LIN {X 0,Y 355.379,Z 611.91,A -85,B 0,C 180,E1 12290.278,E2 12290.278} C_VEL
LIN {X 0,Y 355.45,Z 611.91,A -85,B 0,C 180,E1 12296.376,E2 12296.376} C_VEL
LIN {X 0,Y 355.743,Z 612.609,A -85,B 0,C 180,E1 12302.347,E2 12302.347} C_VEL
LIN {X 0,Y 357.646,Z 617.074,A -85,B 0,C 180,E1 12304.424,E2 12304.424} C_VEL
LIN {X 0,Y 362.835,Z 620.735,A -85,B 0,C 180,E1 12309.929,E2 12309.929} C_VEL
LIN {X 0,Y 365.157,Z 625.028,A -85,B 0,C 180,E1 12313.368,E2 12313.368} C_VEL
LIN {X 0,Y 368.691,Z 627.214,A -85,B 0,C 180,E1 12319.387,E2 12319.387} C_VEL
LIN {X 0,Y 370.662,Z 628.317,A -85,B 0,C 180,E1 12325.314,E2 12325.314} C_VEL
LIN {X 0,Y 371.12,Z 629.145,A -85,B 0,C 180,E1 12330,E2 12330} C_VEL
LIN {X 0,Y 370.62,Z 627.699,A -85,B 0,C 180,E1 12335.127,E2 12335.127} C_VEL
LIN {X 0,Y 368.358,Z 627.102,A -85,B 0,C 180,E1 12341.241,E2 12341.241} C_VEL
LIN {X 0,Y 364.863,Z 624.711,A -85,B 0,C 180,E1 12347.042,E2 12347.042} C_VEL
LIN {X 0,Y 362.708,Z 620.111,A -85,B 0,C 180,E1 12350.279,E2 12350.279} C_VEL
LIN {X 0,Y 357.276,Z 616.633,A -85,B 0,C 180,E1 12355.924,E2 12355.924} C_VEL
LIN {X 0,Y 355.733,Z 612.233,A -85,B 0,C 180,E1 12357.698,E2 12357.698} C_VEL
LIN {X 0,Y 355.573,Z 611.91,A -85,B 0,C 180,E1 12363.611,E2 12363.611} C_VEL
LIN {X 0,Y 355.371,Z 611.91,A -85,B 0,C 180,E1 12369.921,E2 12369.921} C_VEL
LIN {X 0,Y 355.212,Z 611.91,A -85,B 0,C 180,E1 12376.997,E2 12376.997} C_VEL
LIN {X 0,Y 355.407,Z 611.91,A -85,B 0,C 180,E1 12384.038,E2 12384.038} C_VEL
LIN {X 0,Y 355.733,Z 611.91,A -85,B 0,C 180,E1 12392.08,E2 12392.08} C_VEL
LIN {X 0,Y 356.072,Z 611.91,A -85,B 0,C 180,E1 12400.109,E2 12400.109} C_VEL
LIN {X 0,Y 356.301,Z 611.91,A -85,B 0,C 180,E1 12407.784,E2 12407.784} C_VEL
LIN {X 0,Y 356.826,Z 611.91,A -85,B 0,C 180,E1 12415.128,E2 12415.128} C_VEL
LIN {X 0,Y 357.149,Z 611.91,A -85,B 0,C 180,E1 12419.996,E2 12419.996} C_VEL
LIN {X 0,Y 356.648,Z 611.91,A -85,B 0,C 180,E1 12427.312,E2 12427.312} C_VEL
LIN {X 0,Y 356.243,Z 611.91,A -85,B 0,C 180,E1 12434.769,E2 12434.769} C_VEL
LIN {X 0,Y 355.891,Z 611.91,A -85,B 0,C 180,E1 12442.507,E2 12442.507} C_VEL
LIN {X 0,Y 355.712,Z 611.91,A -85,B 0,C 180,E1 12447.912,E2 12447.912} C_VEL
LIN {X 0,Y 355.436,Z 611.91,A -85,B 0,C 180,E1 12455.968,E2 12455.968} C_VEL
LIN {X 0,Y 355.447,Z 612.191,A -85,B 0,C 180,E1 12463.097,E2 12463.097} C_VEL
LIN {X 0,Y 358.002,Z 617.714,A -85,B 0,C 180,E1 12463.686,E2 12463.686} C_VEL
LIN {X 0,Y 377.621,Z 652.126,A -85,B 0,C 180,E1 12467.658,E2 12467.658} C_VEL
LIN {X 0,Y 390.531,Z 683.879,A -85,B 0,C 180,E1 12470.83,E2 12470.83} C_VEL
LIN {X 0,Y 390.809,Z 689.821,A -85,B 0,C 180,E1 12471.237,E2 12471.237} C_VEL
LIN {X 0,Y 385.398,Z 724.931,A -85,B 0,C 180,E1 12473.37,E2 12473.37} C_VEL
LIN {X 0,Y 378.325,Z 760.211,A -85,B 0,C 180,E1 12476.611,E2 12476.611} C_VEL
LIN {X 0,Y 371.725,Z 789.157,A -85,B 0,C 180,E1 12480.406,E2 12480.406} C_VEL
LIN {X 0,Y 365.554,Z 815.678,A -85,B 0,C 180,E1 12485.206,E2 12485.206} C_VEL
LIN {X 0,Y 361.007,Z 837.123,A -85,B 0,C 180,E1 12490.726,E2 12490.726} C_VEL
LIN {X 0,Y 358.596,Z 851.842,A -85,B 0,C 180,E1 12496.164,E2 12496.164} C_VEL
LIN {X 0,Y 357.652,Z 861.108,A -85,B 0,C 180,E1 12501.479,E2 12501.479} C_VEL
LIN {X 0,Y 357.41,Z 864.984,A -85,B 0,C 180,E1 12505.14,E2 12505.14} C_VEL
LIN {X 0,Y 357.395,Z 866.804,A -85,B 0,C 180,E1 12510,E2 12510} C_VEL
LIN {X 0,Y 357.423,Z 864.984,A -85,B 0,C 180,E1 12514.86,E2 12514.86} C_VEL
LIN {X 0,Y 357.893,Z 857.822,A -85,B 0,C 180,E1 12520.716,E2 12520.716} C_VEL
LIN {X 0,Y 359.264,Z 846.967,A -85,B 0,C 180,E1 12525.875,E2 12525.875} C_VEL
LIN {X 0,Y 358.591,Z 843.692,A -85,B 0,C 180,E1 12527.166,E2 12527.166} C_VEL
LIN {X 0,Y 354.052,Z 833.781,A -85,B 0,C 180,E1 12530.653,E2 12530.653} C_VEL
LIN {X 0,Y 354.208,Z 832.758,A -85,B 0,C 180,E1 12530.967,E2 12530.967} C_VEL
LIN {X 0,Y 359.253,Z 810.976,A -85,B 0,C 180,E1 12536.265,E2 12536.265} C_VEL
LIN {X 0,Y 365.983,Z 784.072,A -85,B 0,C 180,E1 12540.966,E2 12540.966} C_VEL
LIN {X 0,Y 373.426,Z 752.301,A -85,B 0,C 180,E1 12544.887,E2 12544.887} C_VEL
LIN {X 0,Y 379.7,Z 721.122,A -85,B 0,C 180,E1 12547.605,E2 12547.605} C_VEL
LIN {X 0,Y 384.344,Z 687.397,A -85,B 0,C 180,E1 12549.682,E2 12549.682} C_VEL
LIN {X 0,Y 372.11,Z 656.453,A -85,B 0,C 180,E1 12552.922,E2 12552.922} C_VEL
LIN {X 0,Y 353.965,Z 623.815,A -85,B 0,C 180,E1 12556.821,E2 12556.821} C_VEL
LIN {X 0,Y 347.602,Z 613.745,A -85,B 0,C 180,E1 12558.246,E2 12558.246} C_VEL
LIN {X 0,Y 347.379,Z 611.91,A -85,B 0,C 180,E1 12558.537,E2 12558.537} C_VEL
LIN {X 0,Y 347.581,Z 611.91,A -85,B 0,C 180,E1 12565.857,E2 12565.857} C_VEL
LIN {X 0,Y 347.709,Z 611.91,A -85,B 0,C 180,E1 12571.388,E2 12571.388} C_VEL
LIN {X 0,Y 348.051,Z 611.91,A -85,B 0,C 180,E1 12579.64,E2 12579.64} C_VEL
LIN {X 0,Y 348.287,Z 611.91,A -85,B 0,C 180,E1 12584.886,E2 12584.886} C_VEL
LIN {X 0,Y 348.726,Z 611.91,A -85,B 0,C 180,E1 12592.521,E2 12592.521} C_VEL
LIN {X 0,Y 349.186,Z 611.91,A -85,B 0,C 180,E1 12600.005,E2 12600.005} C_VEL
LIN {X 0,Y 348.793,Z 611.91,A -85,B 0,C 180,E1 12607.487,E2 12607.487} C_VEL
LIN {X 0,Y 348.3,Z 611.91,A -85,B 0,C 180,E1 12615.123,E2 12615.123} C_VEL
LIN {X 0,Y 348.081,Z 611.91,A -85,B 0,C 180,E1 12620.368,E2 12620.368} C_VEL
LIN {X 0,Y 347.814,Z 611.91,A -85,B 0,C 180,E1 12625.809,E2 12625.809} C_VEL
LIN {X 0,Y 347.611,Z 611.91,A -85,B 0,C 180,E1 12631.516,E2 12631.516} C_VEL
LIN {X 0,Y 347.4,Z 611.91,A -85,B 0,C 180,E1 12638.327,E2 12638.327} C_VEL
LIN {X 0,Y 347.356,Z 611.91,A -85,B 0,C 180,E1 12645.781,E2 12645.781} C_VEL
LIN {X 0,Y 347.391,Z 611.91,A -85,B 0,C 180,E1 12652.398,E2 12652.398} C_VEL
LIN {X 0,Y 347.567,Z 612.488,A -85,B 0,C 180,E1 12656.155,E2 12656.155} C_VEL
LIN {X 0,Y 349.455,Z 617.075,A -85,B 0,C 180,E1 12657.916,E2 12657.916} C_VEL
LIN {X 0,Y 354.366,Z 620.607,A -85,B 0,C 180,E1 12662.05,E2 12662.05} C_VEL
LIN {X 0,Y 357.147,Z 625.381,A -85,B 0,C 180,E1 12664.917,E2 12664.917} C_VEL
LIN {X 0,Y 361.714,Z 628.59,A -85,B 0,C 180,E1 12669.782,E2 12669.782} C_VEL
LIN {X 0,Y 364.262,Z 632.973,A -85,B 0,C 180,E1 12673.475,E2 12673.475} C_VEL
LIN {X 0,Y 367.686,Z 635.044,A -85,B 0,C 180,E1 12679.321,E2 12679.321} C_VEL
LIN {X 0,Y 369.663,Z 636.06,A -85,B 0,C 180,E1 12685.154,E2 12685.154} C_VEL
LIN {X 0,Y 370.158,Z 636.98,A -85,B 0,C 180,E1 12690,E2 12690} C_VEL
LIN {X 0,Y 369.641,Z 635.622,A -85,B 0,C 180,E1 12695.141,E2 12695.141} C_VEL
LIN {X 0,Y 367.366,Z 634.934,A -85,B 0,C 180,E1 12701.289,E2 12701.289} C_VEL
LIN {X 0,Y 363.854,Z 632.55,A -85,B 0,C 180,E1 12707.091,E2 12707.091} C_VEL
LIN {X 0,Y 361.484,Z 627.935,A -85,B 0,C 180,E1 12710.529,E2 12710.529} C_VEL
LIN {X 0,Y 356.027,Z 624.281,A -85,B 0,C 180,E1 12716.169,E2 12716.169} C_VEL
LIN {X 0,Y 353.922,Z 619.616,A -85,B 0,C 180,E1 12718.416,E2 12718.416} C_VEL
LIN {X 0,Y 348.765,Z 616.01,A -85,B 0,C 180,E1 12722.672,E2 12722.672} C_VEL
LIN {X 0,Y 347.632,Z 611.91,A -85,B 0,C 180,E1 12724.151,E2 12724.151} C_VEL
LIN {X 0,Y 347.34,Z 611.91,A -85,B 0,C 180,E1 12730.832,E2 12730.832} C_VEL
LIN {X 0,Y 347.23,Z 611.91,A -85,B 0,C 180,E1 12737.839,E2 12737.839} C_VEL
LIN {X 0,Y 347.499,Z 611.91,A -85,B 0,C 180,E1 12745.876,E2 12745.876} C_VEL
LIN {X 0,Y 347.707,Z 611.91,A -85,B 0,C 180,E1 12751.377,E2 12751.377} C_VEL
LIN {X 0,Y 347.941,Z 611.91,A -85,B 0,C 180,E1 12756.94,E2 12756.94} C_VEL
LIN {X 0,Y 348.23,Z 611.91,A -85,B 0,C 180,E1 12763.044,E2 12763.044} C_VEL
LIN {X 0,Y 348.513,Z 611.91,A -85,B 0,C 180,E1 12769.989,E2 12769.989} C_VEL
LIN {X 0,Y 349.171,Z 611.91,A -85,B 0,C 180,E1 12777.51,E2 12777.51} C_VEL
LIN {X 0,Y 348.959,Z 611.91,A -85,B 0,C 180,E1 12783.698,E2 12783.698} C_VEL
LIN {X 0,Y 348.566,Z 611.91,A -85,B 0,C 180,E1 12790.001,E2 12790.001} C_VEL
LIN {X 0,Y 348.218,Z 611.91,A -85,B 0,C 180,E1 12797.714,E2 12797.714} C_VEL
LIN {X 0,Y 347.81,Z 611.91,A -85,B 0,C 180,E1 12805.799,E2 12805.799} C_VEL
LIN {X 0,Y 347.608,Z 611.91,A -85,B 0,C 180,E1 12811.505,E2 12811.505} C_VEL
LIN {X 0,Y 347.362,Z 611.91,A -85,B 0,C 180,E1 12818.319,E2 12818.319} C_VEL
LIN {X 0,Y 347.385,Z 611.91,A -85,B 0,C 180,E1 12821.624,E2 12821.624} C_VEL
LIN {X 0,Y 349.801,Z 617.549,A -85,B 0,C 180,E1 12822.266,E2 12822.266} C_VEL
LIN {X 0,Y 367.979,Z 648.141,A -85,B 0,C 180,E1 12826.155,E2 12826.155} C_VEL
LIN {X 0,Y 381.568,Z 679.064,A -85,B 0,C 180,E1 12829.463,E2 12829.463} C_VEL
LIN {X 0,Y 384.605,Z 689.979,A -85,B 0,C 180,E1 12830.517,E2 12830.517} C_VEL
LIN {X 0,Y 378.964,Z 724.841,A -85,B 0,C 180,E1 12832.658,E2 12832.658} C_VEL
LIN {X 0,Y 371.582,Z 760.259,A -85,B 0,C 180,E1 12835.961,E2 12835.961} C_VEL
LIN {X 0,Y 364.719,Z 788.918,A -85,B 0,C 180,E1 12839.779,E2 12839.779} C_VEL
LIN {X 0,Y 358.241,Z 815.44,A -85,B 0,C 180,E1 12844.664,E2 12844.664} C_VEL
LIN {X 0,Y 353.23,Z 837.693,A -85,B 0,C 180,E1 12850.54,E2 12850.54} C_VEL
LIN {X 0,Y 350.78,Z 851.604,A -85,B 0,C 180,E1 12855.849,E2 12855.849} C_VEL
LIN {X 0,Y 349.761,Z 860.872,A -85,B 0,C 180,E1 12861.286,E2 12861.286} C_VEL
LIN {X 0,Y 349.527,Z 864.75,A -85,B 0,C 180,E1 12865.03,E2 12865.03} C_VEL
LIN {X 0,Y 349.497,Z 866.57,A -85,B 0,C 180,E1 12870,E2 12870} C_VEL
LIN {X 0,Y 349.535,Z 864.703,A -85,B 0,C 180,E1 12875.027,E2 12875.027} C_VEL
LIN {X 0,Y 350.085,Z 857.155,A -85,B 0,C 180,E1 12881.222,E2 12881.222} C_VEL
LIN {X 0,Y 351.825,Z 845.129,A -85,B 0,C 180,E1 12886.887,E2 12886.887} C_VEL
LIN {X 0,Y 354.208,Z 832.758,A -85,B 0,C 180,E1 12890.967,E2 12890.967} C_VEL
LIN {X 0,Y 353.966,Z 828.625,A -85,B 0,C 180,E1 12892.216,E2 12892.216} C_VEL
LIN {X 0,Y 350.612,Z 816.511,A -85,B 0,C 180,E1 12895.591,E2 12895.591} C_VEL
LIN {X 0,Y 350.885,Z 815.282,A -85,B 0,C 180,E1 12895.884,E2 12895.884} C_VEL
LIN {X 0,Y 357.75,Z 788.679,A -85,B 0,C 180,E1 12900.874,E2 12900.874} C_VEL
LIN {X 0,Y 364.953,Z 760.3,A -85,B 0,C 180,E1 12904.708,E2 12904.708} C_VEL
LIN {X 0,Y 372.322,Z 726.203,A -85,B 0,C 180,E1 12907.956,E2 12907.956} C_VEL
LIN {X 0,Y 378.078,Z 690.576,A -85,B 0,C 180,E1 12910.247,E2 12910.247} C_VEL
LIN {X 0,Y 366.369,Z 660.181,A -85,B 0,C 180,E1 12913.582,E2 12913.582} C_VEL
LIN {X 0,Y 349.756,Z 629.585,A -85,B 0,C 180,E1 12917.384,E2 12917.384} C_VEL
LIN {X 0,Y 339.555,Z 613.362,A -85,B 0,C 180,E1 12919.791,E2 12919.791} C_VEL
LIN {X 0,Y 339.435,Z 611.91,A -85,B 0,C 180,E1 12920.003,E2 12920.003} C_VEL
LIN {X 0,Y 339.666,Z 611.91,A -85,B 0,C 180,E1 12927.878,E2 12927.878} C_VEL
LIN {X 0,Y 339.801,Z 611.91,A -85,B 0,C 180,E1 12933.546,E2 12933.546} C_VEL
LIN {X 0,Y 340.23,Z 611.91,A -85,B 0,C 180,E1 12941.856,E2 12941.856} C_VEL
LIN {X 0,Y 340.628,Z 611.91,A -85,B 0,C 180,E1 12949.764,E2 12949.764} C_VEL
LIN {X 0,Y 341.156,Z 611.91,A -85,B 0,C 180,E1 12957.461,E2 12957.461} C_VEL
LIN {X 0,Y 341.262,Z 611.91,A -85,B 0,C 180,E1 12962.547,E2 12962.547} C_VEL
LIN {X 0,Y 340.616,Z 611.91,A -85,B 0,C 180,E1 12970.246,E2 12970.246} C_VEL
LIN {X 0,Y 340.252,Z 611.91,A -85,B 0,C 180,E1 12978.153,E2 12978.153} C_VEL
LIN {X 0,Y 339.809,Z 611.91,A -85,B 0,C 180,E1 12986.463,E2 12986.463} C_VEL
LIN {X 0,Y 339.634,Z 611.91,A -85,B 0,C 180,E1 12992.344,E2 12992.344} C_VEL
LIN {X 0,Y 339.463,Z 611.91,A -85,B 0,C 180,E1 13000.692,E2 13000.692} C_VEL
LIN {X 0,Y 339.446,Z 611.91,A -85,B 0,C 180,E1 13008.006,E2 13008.006} C_VEL
LIN {X 0,Y 339.46,Z 612.679,A -85,B 0,C 180,E1 13010.86,E2 13010.86} C_VEL
LIN {X 0,Y 341.535,Z 617.232,A -85,B 0,C 180,E1 13012.536,E2 13012.536} C_VEL
LIN {X 0,Y 346.1,Z 620.708,A -85,B 0,C 180,E1 13015.866,E2 13015.866} C_VEL
LIN {X 0,Y 349.099,Z 625.579,A -85,B 0,C 180,E1 13018.458,E2 13018.458} C_VEL
LIN {X 0,Y 353.078,Z 628.56,A -85,B 0,C 180,E1 13021.814,E2 13021.814} C_VEL
LIN {X 0,Y 356.3,Z 633.388,A -85,B 0,C 180,E1 13025.062,E2 13025.062} C_VEL
LIN {X 0,Y 360.55,Z 636.426,A -85,B 0,C 180,E1 13029.595,E2 13029.595} C_VEL
LIN {X 0,Y 363.477,Z 641.06,A -85,B 0,C 180,E1 13033.738,E2 13033.738} C_VEL
LIN {X 0,Y 366.703,Z 642.866,A -85,B 0,C 180,E1 13039.292,E2 13039.292} C_VEL
LIN {X 0,Y 368.684,Z 643.989,A -85,B 0,C 180,E1 13045.141,E2 13045.141} C_VEL
LIN {X 0,Y 369.195,Z 644.82,A -85,B 0,C 180,E1 13050,E2 13050} C_VEL
LIN {X 0,Y 368.647,Z 643.398,A -85,B 0,C 180,E1 13055.302,E2 13055.302} C_VEL
LIN {X 0,Y 366.384,Z 642.769,A -85,B 0,C 180,E1 13061.32,E2 13061.32} C_VEL
LIN {X 0,Y 362.845,Z 640.388,A -85,B 0,C 180,E1 13067.139,E2 13067.139} C_VEL
LIN {X 0,Y 360.263,Z 635.571,A -85,B 0,C 180,E1 13070.811,E2 13070.811} C_VEL
LIN {X 0,Y 354.847,Z 631.993,A -85,B 0,C 180,E1 13076.354,E2 13076.354} C_VEL
LIN {X 0,Y 352.387,Z 627.308,A -85,B 0,C 180,E1 13078.899,E2 13078.899} C_VEL
LIN {X 0,Y 347.225,Z 623.305,A -85,B 0,C 180,E1 13083.102,E2 13083.102} C_VEL
LIN {X 0,Y 345.338,Z 619.491,A -85,B 0,C 180,E1 13084.747,E2 13084.747} C_VEL
LIN {X 0,Y 340.583,Z 615.849,A -85,B 0,C 180,E1 13088.181,E2 13088.181} C_VEL
LIN {X 0,Y 339.401,Z 611.91,A -85,B 0,C 180,E1 13089.402,E2 13089.402} C_VEL
LIN {X 0,Y 339.346,Z 611.91,A -85,B 0,C 180,E1 13095.55,E2 13095.55} C_VEL
LIN {X 0,Y 339.358,Z 611.91,A -85,B 0,C 180,E1 13103.425,E2 13103.425} C_VEL
LIN {X 0,Y 339.749,Z 611.91,A -85,B 0,C 180,E1 13110.642,E2 13110.642} C_VEL
LIN {X 0,Y 340.155,Z 611.91,A -85,B 0,C 180,E1 13119.184,E2 13119.184} C_VEL
LIN {X 0,Y 340.398,Z 611.91,A -85,B 0,C 180,E1 13127.146,E2 13127.146} C_VEL
LIN {X 0,Y 341.004,Z 611.91,A -85,B 0,C 180,E1 13134.901,E2 13134.901} C_VEL
LIN {X 0,Y 341.357,Z 611.91,A -85,B 0,C 180,E1 13139.995,E2 13139.995} C_VEL
LIN {X 0,Y 340.79,Z 611.91,A -85,B 0,C 180,E1 13147.654,E2 13147.654} C_VEL
LIN {X 0,Y 340.363,Z 611.91,A -85,B 0,C 180,E1 13155.475,E2 13155.475} C_VEL
LIN {X 0,Y 340.107,Z 611.91,A -85,B 0,C 180,E1 13160.857,E2 13160.857} C_VEL
LIN {X 0,Y 339.739,Z 611.91,A -85,B 0,C 180,E1 13169.348,E2 13169.348} C_VEL
LIN {X 0,Y 339.405,Z 611.91,A -85,B 0,C 180,E1 13176.586,E2 13176.586} C_VEL
LIN {X 0,Y 339.442,Z 612.101,A -85,B 0,C 180,E1 13180.146,E2 13180.146} C_VEL
LIN {X 0,Y 341.796,Z 617.496,A -85,B 0,C 180,E1 13180.778,E2 13180.778} C_VEL
LIN {X 0,Y 359.45,Z 646.383,A -85,B 0,C 180,E1 13184.787,E2 13184.787} C_VEL
LIN {X 0,Y 373.569,Z 677.202,A -85,B 0,C 180,E1 13188.32,E2 13188.32} C_VEL
LIN {X 0,Y 378.14,Z 692.296,A -85,B 0,C 180,E1 13189.875,E2 13189.875} C_VEL
LIN {X 0,Y 372.313,Z 726.204,A -85,B 0,C 180,E1 13192.043,E2 13192.043} C_VEL
LIN {X 0,Y 364.714,Z 761.114,A -85,B 0,C 180,E1 13195.375,E2 13195.375} C_VEL
LIN {X 0,Y 357.274,Z 790.577,A -85,B 0,C 180,E1 13199.434,E2 13199.434} C_VEL
LIN {X 0,Y 350.943,Z 815.2,A -85,B 0,C 180,E1 13204.099,E2 13204.099} C_VEL
LIN {X 0,Y 345.595,Z 837.453,A -85,B 0,C 180,E1 13210.092,E2 13210.092} C_VEL
LIN {X 0,Y 342.957,Z 851.56,A -85,B 0,C 180,E1 13215.619,E2 13215.619} C_VEL
LIN {X 0,Y 341.884,Z 860.637,A -85,B 0,C 180,E1 13221.083,E2 13221.083} C_VEL
LIN {X 0,Y 341.663,Z 864.517,A -85,B 0,C 180,E1 13224.915,E2 13224.915} C_VEL
LIN {X 0,Y 341.623,Z 866.338,A -85,B 0,C 180,E1 13230,E2 13230} C_VEL
LIN {X 0,Y 341.663,Z 864.517,A -85,B 0,C 180,E1 13235.085,E2 13235.085} C_VEL
LIN {X 0,Y 342.129,Z 857.947,A -85,B 0,C 180,E1 13240.841,E2 13240.841} C_VEL
LIN {X 0,Y 344.11,Z 844.89,A -85,B 0,C 180,E1 13247.277,E2 13247.277} C_VEL
LIN {X 0,Y 348.318,Z 825.42,A -85,B 0,C 180,E1 13253.416,E2 13253.416} C_VEL
LIN {X 0,Y 350.885,Z 815.282,A -85,B 0,C 180,E1 13255.884,E2 13255.884} C_VEL
LIN {X 0,Y 349.952,Z 805.507,A -85,B 0,C 180,E1 13258.261,E2 13258.261} C_VEL
LIN {X 0,Y 349.169,Z 794.676,A -85,B 0,C 180,E1 13260.523,E2 13260.523} C_VEL
LIN {X 0,Y 357.221,Z 764.533,A -85,B 0,C 180,E1 13264.903,E2 13264.903} C_VEL
LIN {X 0,Y 364.571,Z 732.849,A -85,B 0,C 180,E1 13268.163,E2 13268.163} C_VEL
LIN {X 0,Y 371.476,Z 696.249,A -85,B 0,C 180,E1 13270.702,E2 13270.702} C_VEL
LIN {X 0,Y 370.264,Z 688.741,A -85,B 0,C 180,E1 13271.384,E2 13271.384} C_VEL
LIN {X 0,Y 358.096,Z 658.476,A -85,B 0,C 180,E1 13274.92,E2 13274.92} C_VEL
LIN {X 0,Y 342.055,Z 629.861,A -85,B 0,C 180,E1 13278.787,E2 13278.787} C_VEL
LIN {X 0,Y 331.735,Z 613.654,A -85,B 0,C 180,E1 13281.394,E2 13281.394} C_VEL
LIN {X 0,Y 331.542,Z 611.91,A -85,B 0,C 180,E1 13281.709,E2 13281.709} C_VEL
LIN {X 0,Y 331.806,Z 611.91,A -85,B 0,C 180,E1 13290.11,E2 13290.11} C_VEL
LIN {X 0,Y 332.076,Z 611.91,A -85,B 0,C 180,E1 13298.614,E2 13298.614} C_VEL
LIN {X 0,Y 332.393,Z 611.91,A -85,B 0,C 180,E1 13304.145,E2 13304.145} C_VEL
LIN {X 0,Y 332.868,Z 611.91,A -85,B 0,C 180,E1 13312.162,E2 13312.162} C_VEL
LIN {X 0,Y 333.397,Z 611.91,A -85,B 0,C 180,E1 13320.005,E2 13320.005} C_VEL
LIN {X 0,Y 333.079,Z 611.91,A -85,B 0,C 180,E1 13325.221,E2 13325.221} C_VEL
LIN {X 0,Y 332.519,Z 611.91,A -85,B 0,C 180,E1 13333.164,E2 13333.164} C_VEL
LIN {X 0,Y 332.274,Z 611.91,A -85,B 0,C 180,E1 13338.605,E2 13338.605} C_VEL
LIN {X 0,Y 331.868,Z 611.91,A -85,B 0,C 180,E1 13347.148,E2 13347.148} C_VEL
LIN {X 0,Y 331.55,Z 611.91,A -85,B 0,C 180,E1 13354.716,E2 13354.716} C_VEL
LIN {X 0,Y 331.531,Z 611.91,A -85,B 0,C 180,E1 13359.748,E2 13359.748} C_VEL
LIN {X 0,Y 331.549,Z 612.641,A -85,B 0,C 180,E1 13366.109,E2 13366.109} C_VEL
LIN {X 0,Y 333.579,Z 617.239,A -85,B 0,C 180,E1 13367.642,E2 13367.642} C_VEL
LIN {X 0,Y 337.838,Z 620.701,A -85,B 0,C 180,E1 13370.488,E2 13370.488} C_VEL
LIN {X 0,Y 341.465,Z 626.057,A -85,B 0,C 180,E1 13373.213,E2 13373.213} C_VEL
LIN {X 0,Y 344.662,Z 628.507,A -85,B 0,C 180,E1 13375.566,E2 13375.566} C_VEL
LIN {X 0,Y 348.217,Z 633.563,A -85,B 0,C 180,E1 13378.549,E2 13378.549} C_VEL
LIN {X 0,Y 351.779,Z 636.249,A -85,B 0,C 180,E1 13381.532,E2 13381.532} C_VEL
LIN {X 0,Y 355.14,Z 641.116,A -85,B 0,C 180,E1 13384.87,E2 13384.87} C_VEL
LIN {X 0,Y 359.349,Z 644.104,A -85,B 0,C 180,E1 13389.344,E2 13389.344} C_VEL
LIN {X 0,Y 362.26,Z 648.7,A -85,B 0,C 180,E1 13393.415,E2 13393.415} C_VEL
LIN {X 0,Y 365.719,Z 650.702,A -85,B 0,C 180,E1 13399.263,E2 13399.263} C_VEL
LIN {X 0,Y 367.686,Z 651.751,A -85,B 0,C 180,E1 13404.98,E2 13404.98} C_VEL
LIN {X 0,Y 368.233,Z 652.66,A -85,B 0,C 180,E1 13410,E2 13410} C_VEL
LIN {X 0,Y 367.668,Z 651.328,A -85,B 0,C 180,E1 13415.316,E2 13415.316} C_VEL
LIN {X 0,Y 365.402,Z 650.604,A -85,B 0,C 180,E1 13421.351,E2 13421.351} C_VEL
LIN {X 0,Y 361.785,Z 648.175,A -85,B 0,C 180,E1 13427.264,E2 13427.264} C_VEL
LIN {X 0,Y 358.181,Z 642.833,A -85,B 0,C 180,E1 13432.053,E2 13432.053} C_VEL
LIN {X 0,Y 353.081,Z 638.832,A -85,B 0,C 180,E1 13437.164,E2 13437.164} C_VEL
LIN {X 0,Y 350.696,Z 634.887,A -85,B 0,C 180,E1 13439.451,E2 13439.451} C_VEL
LIN {X 0,Y 345.68,Z 630.569,A -85,B 0,C 180,E1 13443.555,E2 13443.555} C_VEL
LIN {X 0,Y 344.157,Z 627.264,A -85,B 0,C 180,E1 13444.884,E2 13444.884} C_VEL
LIN {X 0,Y 339.11,Z 623.354,A -85,B 0,C 180,E1 13448.526,E2 13448.526} C_VEL
LIN {X 0,Y 336.94,Z 619.418,A -85,B 0,C 180,E1 13450.186,E2 13450.186} C_VEL
LIN {X 0,Y 332.177,Z 615.326,A -85,B 0,C 180,E1 13453.329,E2 13453.329} C_VEL
LIN {X 0,Y 331.442,Z 611.91,A -85,B 0,C 180,E1 13454.287,E2 13454.287} C_VEL
LIN {X 0,Y 331.414,Z 611.91,A -85,B 0,C 180,E1 13460.954,E2 13460.954} C_VEL
LIN {X 0,Y 331.548,Z 611.91,A -85,B 0,C 180,E1 13466.766,E2 13466.766} C_VEL
LIN {X 0,Y 331.888,Z 611.91,A -85,B 0,C 180,E1 13472.854,E2 13472.854} C_VEL
LIN {X 0,Y 332.16,Z 611.91,A -85,B 0,C 180,E1 13478.609,E2 13478.609} C_VEL
LIN {X 0,Y 332.359,Z 611.91,A -85,B 0,C 180,E1 13484.133,E2 13484.133} C_VEL
LIN {X 0,Y 332.902,Z 611.91,A -85,B 0,C 180,E1 13492.154,E2 13492.154} C_VEL
LIN {X 0,Y 333.453,Z 611.91,A -85,B 0,C 180,E1 13499.995,E2 13499.995} C_VEL
LIN {X 0,Y 332.868,Z 611.91,A -85,B 0,C 180,E1 13507.838,E2 13507.838} C_VEL
LIN {X 0,Y 332.4,Z 611.91,A -85,B 0,C 180,E1 13515.855,E2 13515.855} C_VEL
LIN {X 0,Y 331.96,Z 611.91,A -85,B 0,C 180,E1 13524.19,E2 13524.19} C_VEL
LIN {X 0,Y 331.754,Z 611.91,A -85,B 0,C 180,E1 13530.127,E2 13530.127} C_VEL
LIN {X 0,Y 331.508,Z 611.91,A -85,B 0,C 180,E1 13538.459,E2 13538.459} C_VEL
LIN {X 0,Y 333.936,Z 617.62,A -85,B 0,C 180,E1 13539.204,E2 13539.204} C_VEL
LIN {X 0,Y 351.594,Z 645.635,A -85,B 0,C 180,E1 13543.467,E2 13543.467} C_VEL
LIN {X 0,Y 366.009,Z 676.532,A -85,B 0,C 180,E1 13547.236,E2 13547.236} C_VEL
LIN {X 0,Y 371.727,Z 694.718,A -85,B 0,C 180,E1 13549.219,E2 13549.219} C_VEL
LIN {X 0,Y 364.971,Z 730.952,A -85,B 0,C 180,E1 13551.681,E2 13551.681} C_VEL
LIN {X 0,Y 357.467,Z 763.335,A -85,B 0,C 180,E1 13554.94,E2 13554.94} C_VEL
LIN {X 0,Y 349.489,Z 793.56,A -85,B 0,C 180,E1 13559.292,E2 13559.292} C_VEL
LIN {X 0,Y 342.897,Z 817.622,A -85,B 0,C 180,E1 13564.148,E2 13564.148} C_VEL
LIN {X 0,Y 337.873,Z 837.791,A -85,B 0,C 180,E1 13569.809,E2 13569.809} C_VEL
LIN {X 0,Y 334.916,Z 852.773,A -85,B 0,C 180,E1 13576.029,E2 13576.029} C_VEL
LIN {X 0,Y 333.881,Z 861.987,A -85,B 0,C 180,E1 13582.181,E2 13582.181} C_VEL
LIN {X 0,Y 333.647,Z 865.648,A -85,B 0,C 180,E1 13587.399,E2 13587.399} C_VEL
LIN {X 0,Y 333.662,Z 865.648,A -85,B 0,C 180,E1 13592.601,E2 13592.601} C_VEL
LIN {X 0,Y 333.878,Z 861.987,A -85,B 0,C 180,E1 13597.819,E2 13597.819} C_VEL
LIN {X 0,Y 334.929,Z 852.741,A -85,B 0,C 180,E1 13603.988,E2 13603.988} C_VEL
LIN {X 0,Y 337.803,Z 838.073,A -85,B 0,C 180,E1 13610.101,E2 13610.101} C_VEL
LIN {X 0,Y 343.289,Z 816.157,A -85,B 0,C 180,E1 13616.207,E2 13616.207} C_VEL
LIN {X 0,Y 349.169,Z 794.676,A -85,B 0,C 180,E1 13620.523,E2 13620.523} C_VEL
LIN {X 0,Y 348.974,Z 783.268,A -85,B 0,C 180,E1 13622.708,E2 13622.708} C_VEL
LIN {X 0,Y 348.762,Z 771.138,A -85,B 0,C 180,E1 13624.788,E2 13624.788} C_VEL
LIN {X 0,Y 357.405,Z 736.839,A -85,B 0,C 180,E1 13628.59,E2 13628.59} C_VEL
LIN {X 0,Y 364.616,Z 701.227,A -85,B 0,C 180,E1 13631.198,E2 13631.198} C_VEL
LIN {X 0,Y 364.932,Z 694.63,A -85,B 0,C 180,E1 13631.696,E2 13631.696} C_VEL
LIN {X 0,Y 353.53,Z 664.276,A -85,B 0,C 180,E1 13635.37,E2 13635.37} C_VEL
LIN {X 0,Y 338.102,Z 635.829,A -85,B 0,C 180,E1 13639.361,E2 13639.361} C_VEL
LIN {X 0,Y 325.956,Z 617.536,A -85,B 0,C 180,E1 13642.538,E2 13642.538} C_VEL
LIN {X 0,Y 323.648,Z 611.91,A -85,B 0,C 180,E1 13643.433,E2 13643.433} C_VEL
LIN {X 0,Y 323.737,Z 611.91,A -85,B 0,C 180,E1 13649.046,E2 13649.046} C_VEL
LIN {X 0,Y 323.938,Z 611.91,A -85,B 0,C 180,E1 13655.131,E2 13655.131} C_VEL
LIN {X 0,Y 324.265,Z 611.91,A -85,B 0,C 180,E1 13660.929,E2 13660.929} C_VEL
LIN {X 0,Y 324.751,Z 611.91,A -85,B 0,C 180,E1 13669.257,E2 13669.257} C_VEL
LIN {X 0,Y 325.351,Z 611.91,A -85,B 0,C 180,E1 13677.338,E2 13677.338} C_VEL
LIN {X 0,Y 325.431,Z 611.91,A -85,B 0,C 180,E1 13682.671,E2 13682.671} C_VEL
LIN {X 0,Y 324.729,Z 611.91,A -85,B 0,C 180,E1 13690.753,E2 13690.753} C_VEL
LIN {X 0,Y 324.473,Z 611.91,A -85,B 0,C 180,E1 13696.263,E2 13696.263} C_VEL
LIN {X 0,Y 324.11,Z 611.91,A -85,B 0,C 180,E1 13701.949,E2 13701.949} C_VEL
LIN {X 0,Y 323.88,Z 611.91,A -85,B 0,C 180,E1 13707.875,E2 13707.875} C_VEL
LIN {X 0,Y 323.639,Z 611.91,A -85,B 0,C 180,E1 13714.156,E2 13714.156} C_VEL
LIN {X 0,Y 323.513,Z 612.547,A -85,B 0,C 180,E1 13721.593,E2 13721.593} C_VEL
LIN {X 0,Y 325.727,Z 617.296,A -85,B 0,C 180,E1 13723.148,E2 13723.148} C_VEL
LIN {X 0,Y 329.773,Z 620.556,A -85,B 0,C 180,E1 13725.664,E2 13725.664} C_VEL
LIN {X 0,Y 333.143,Z 625.759,A -85,B 0,C 180,E1 13728.027,E2 13728.027} C_VEL
LIN {X 0,Y 336.35,Z 628.567,A -85,B 0,C 180,E1 13730.178,E2 13730.178} C_VEL
LIN {X 0,Y 340.701,Z 634.098,A -85,B 0,C 180,E1 13733.386,E2 13733.386} C_VEL
LIN {X 0,Y 343.308,Z 636.309,A -85,B 0,C 180,E1 13735.319,E2 13735.319} C_VEL
LIN {X 0,Y 347.216,Z 641.445,A -85,B 0,C 180,E1 13738.542,E2 13738.542} C_VEL
LIN {X 0,Y 350.572,Z 644.114,A -85,B 0,C 180,E1 13741.34,E2 13741.34} C_VEL
LIN {X 0,Y 354.404,Z 649.173,A -85,B 0,C 180,E1 13745.128,E2 13745.128} C_VEL
LIN {X 0,Y 358.288,Z 652.003,A -85,B 0,C 180,E1 13749.261,E2 13749.261} C_VEL
LIN {X 0,Y 361.406,Z 656.666,A -85,B 0,C 180,E1 13753.574,E2 13753.574} C_VEL
LIN {X 0,Y 364.735,Z 658.538,A -85,B 0,C 180,E1 13759.234,E2 13759.234} C_VEL
LIN {X 0,Y 366.715,Z 659.614,A -85,B 0,C 180,E1 13764.967,E2 13764.967} C_VEL
LIN {X 0,Y 367.27,Z 660.5,A -85,B 0,C 180,E1 13770,E2 13770} C_VEL
LIN {X 0,Y 366.659,Z 659.016,A -85,B 0,C 180,E1 13775.629,E2 13775.629} C_VEL
LIN {X 0,Y 364.15,Z 658.278,A -85,B 0,C 180,E1 13781.999,E2 13781.999} C_VEL
LIN {X 0,Y 360.313,Z 655.481,A -85,B 0,C 180,E1 13788.02,E2 13788.02} C_VEL
LIN {X 0,Y 357.5,Z 650.726,A -85,B 0,C 180,E1 13791.773,E2 13791.773} C_VEL
LIN {X 0,Y 352.119,Z 646.908,A -85,B 0,C 180,E1 13797.125,E2 13797.125} C_VEL
LIN {X 0,Y 349.582,Z 642.669,A -85,B 0,C 180,E1 13799.554,E2 13799.554} C_VEL
LIN {X 0,Y 344.411,Z 638.275,A -85,B 0,C 180,E1 13803.777,E2 13803.777} C_VEL
LIN {X 0,Y 342.361,Z 634.87,A -85,B 0,C 180,E1 13805.469,E2 13805.469} C_VEL
LIN {X 0,Y 337.246,Z 630.296,A -85,B 0,C 180,E1 13809.122,E2 13809.122} C_VEL
LIN {X 0,Y 335.26,Z 627,A -85,B 0,C 180,E1 13810.604,E2 13810.604} C_VEL
LIN {X 0,Y 330.379,Z 622.387,A -85,B 0,C 180,E1 13813.846,E2 13813.846} C_VEL
LIN {X 0,Y 328.948,Z 619.428,A -85,B 0,C 180,E1 13814.881,E2 13814.881} C_VEL
LIN {X 0,Y 324.084,Z 615.196,A -85,B 0,C 180,E1 13817.906,E2 13817.906} C_VEL
LIN {X 0,Y 323.369,Z 611.91,A -85,B 0,C 180,E1 13818.776,E2 13818.776} C_VEL
LIN {X 0,Y 323.586,Z 611.91,A -85,B 0,C 180,E1 13825.838,E2 13825.838} C_VEL
LIN {X 0,Y 323.946,Z 611.91,A -85,B 0,C 180,E1 13832.625,E2 13832.625} C_VEL
LIN {X 0,Y 324.306,Z 611.91,A -85,B 0,C 180,E1 13840.921,E2 13840.921} C_VEL
LIN {X 0,Y 324.675,Z 611.91,A -85,B 0,C 180,E1 13849.245,E2 13849.245} C_VEL
LIN {X 0,Y 325.431,Z 611.91,A -85,B 0,C 180,E1 13857.329,E2 13857.329} C_VEL
LIN {X 0,Y 325.359,Z 611.91,A -85,B 0,C 180,E1 13862.662,E2 13862.662} C_VEL
LIN {X 0,Y 324.75,Z 611.91,A -85,B 0,C 180,E1 13870.743,E2 13870.743} C_VEL
LIN {X 0,Y 324.288,Z 611.91,A -85,B 0,C 180,E1 13879.07,E2 13879.07} C_VEL
LIN {X 0,Y 323.937,Z 611.91,A -85,B 0,C 180,E1 13887.372,E2 13887.372} C_VEL
LIN {X 0,Y 323.588,Z 611.91,A -85,B 0,C 180,E1 13895.686,E2 13895.686} C_VEL
LIN {X 0,Y 323.605,Z 612.094,A -85,B 0,C 180,E1 13896.723,E2 13896.723} C_VEL
LIN {X 0,Y 325.951,Z 617.569,A -85,B 0,C 180,E1 13897.462,E2 13897.462} C_VEL
LIN {X 0,Y 339.268,Z 637.755,A -85,B 0,C 180,E1 13900.938,E2 13900.938} C_VEL
LIN {X 0,Y 354.291,Z 665.861,A -85,B 0,C 180,E1 13904.831,E2 13904.831} C_VEL
LIN {X 0,Y 365.398,Z 696.011,A -85,B 0,C 180,E1 13908.473,E2 13908.473} C_VEL
LIN {X 0,Y 358.098,Z 733.705,A -85,B 0,C 180,E1 13911.14,E2 13911.14} C_VEL
LIN {X 0,Y 350.234,Z 765.488,A -85,B 0,C 180,E1 13914.486,E2 13914.486} C_VEL
LIN {X 0,Y 342.392,Z 793.893,A -85,B 0,C 180,E1 13918.696,E2 13918.696} C_VEL
LIN {X 0,Y 335.143,Z 819.087,A -85,B 0,C 180,E1 13923.965,E2 13923.965} C_VEL
LIN {X 0,Y 330.342,Z 837.22,A -85,B 0,C 180,E1 13929.215,E2 13929.215} C_VEL
LIN {X 0,Y 327.238,Z 851.727,A -85,B 0,C 180,E1 13935.259,E2 13935.259} C_VEL
LIN {X 0,Y 326.14,Z 860.166,A -85,B 0,C 180,E1 13940.649,E2 13940.649} C_VEL
LIN {X 0,Y 325.88,Z 864.049,A -85,B 0,C 180,E1 13944.668,E2 13944.668} C_VEL
LIN {X 0,Y 325.828,Z 865.871,A -85,B 0,C 180,E1 13950,E2 13950} C_VEL
LIN {X 0,Y 325.88,Z 864.049,A -85,B 0,C 180,E1 13955.332,E2 13955.332} C_VEL
LIN {X 0,Y 326.435,Z 857.474,A -85,B 0,C 180,E1 13961.369,E2 13961.369} C_VEL
LIN {X 0,Y 328.696,Z 844.412,A -85,B 0,C 180,E1 13968.115,E2 13968.115} C_VEL
LIN {X 0,Y 333.53,Z 824.848,A -85,B 0,C 180,E1 13974.549,E2 13974.549} C_VEL
LIN {X 0,Y 339.883,Z 802.469,A -85,B 0,C 180,E1 13979.706,E2 13979.706} C_VEL
LIN {X 0,Y 348.059,Z 773.777,A -85,B 0,C 180,E1 13984.437,E2 13984.437} C_VEL
LIN {X 0,Y 348.762,Z 771.138,A -85,B 0,C 180,E1 13984.788,E2 13984.788} C_VEL
LIN {X 0,Y 348.911,Z 758.297,A -85,B 0,C 180,E1 13986.756,E2 13986.756} C_VEL
LIN {X 0,Y 349.16,Z 744.852,A -85,B 0,C 180,E1 13988.597,E2 13988.597} C_VEL
LIN {X 0,Y 357.208,Z 709.169,A -85,B 0,C 180,E1 13991.536,E2 13991.536} C_VEL
LIN {X 0,Y 358.575,Z 697.275,A -85,B 0,C 180,E1 13992.368,E2 13992.368} C_VEL
LIN {X 0,Y 347.178,Z 666.552,A -85,B 0,C 180,E1 13996.303,E2 13996.303} C_VEL
LIN {X 0,Y 332.885,Z 639.999,A -85,B 0,C 180,E1 14000.246,E2 14000.246} C_VEL
LIN {X 0,Y 318.422,Z 617.818,A -85,B 0,C 180,E1 14004.32,E2 14004.32} C_VEL
LIN {X 0,Y 315.789,Z 612.869,A -85,B 0,C 180,E1 14005.177,E2 14005.177} C_VEL
LIN {X 0,Y 315.765,Z 611.91,A -85,B 0,C 180,E1 14005.659,E2 14005.659} C_VEL
LIN {X 0,Y 315.859,Z 611.91,A -85,B 0,C 180,E1 14011.364,E2 14011.364} C_VEL
LIN {X 0,Y 316.085,Z 611.91,A -85,B 0,C 180,E1 14017.474,E2 14017.474} C_VEL
LIN {X 0,Y 316.474,Z 611.91,A -85,B 0,C 180,E1 14023.325,E2 14023.325} C_VEL
LIN {X 0,Y 316.988,Z 611.91,A -85,B 0,C 180,E1 14031.767,E2 14031.767} C_VEL
LIN {X 0,Y 317.614,Z 611.91,A -85,B 0,C 180,E1 14040.005,E2 14040.005} C_VEL
LIN {X 0,Y 317.236,Z 611.91,A -85,B 0,C 180,E1 14045.482,E2 14045.482} C_VEL
LIN {X 0,Y 316.631,Z 611.91,A -85,B 0,C 180,E1 14053.837,E2 14053.837} C_VEL
LIN {X 0,Y 316.342,Z 611.91,A -85,B 0,C 180,E1 14059.579,E2 14059.579} C_VEL
LIN {X 0,Y 316.018,Z 611.91,A -85,B 0,C 180,E1 14065.548,E2 14065.548} C_VEL
LIN {X 0,Y 315.74,Z 611.91,A -85,B 0,C 180,E1 14071.84,E2 14071.84} C_VEL
LIN {X 0,Y 315.704,Z 612.062,A -85,B 0,C 180,E1 14077.523,E2 14077.523} C_VEL
LIN {X 0,Y 317.121,Z 616.65,A -85,B 0,C 180,E1 14078.51,E2 14078.51} C_VEL
LIN {X 0,Y 321.648,Z 620.492,A -85,B 0,C 180,E1 14081.136,E2 14081.136} C_VEL
LIN {X 0,Y 325.394,Z 625.869,A -85,B 0,C 180,E1 14083.578,E2 14083.578} C_VEL
LIN {X 0,Y 328.129,Z 628.281,A -85,B 0,C 180,E1 14085.3,E2 14085.3} C_VEL
LIN {X 0,Y 332.298,Z 633.802,A -85,B 0,C 180,E1 14088.135,E2 14088.135} C_VEL
LIN {X 0,Y 334.964,Z 636.402,A -85,B 0,C 180,E1 14089.929,E2 14089.929} C_VEL
LIN {X 0,Y 339.666,Z 641.964,A -85,B 0,C 180,E1 14093.359,E2 14093.359} C_VEL
LIN {X 0,Y 342.006,Z 644.22,A -85,B 0,C 180,E1 14095.111,E2 14095.111} C_VEL
LIN {X 0,Y 346.474,Z 649.472,A -85,B 0,C 180,E1 14098.741,E2 14098.741} C_VEL
LIN {X 0,Y 349.4,Z 652.061,A -85,B 0,C 180,E1 14101.192,E2 14101.192} C_VEL
LIN {X 0,Y 353.565,Z 657.145,A -85,B 0,C 180,E1 14105.275,E2 14105.275} C_VEL
LIN {X 0,Y 357.176,Z 659.826,A -85,B 0,C 180,E1 14109.113,E2 14109.113} C_VEL
LIN {X 0,Y 360.275,Z 664.397,A -85,B 0,C 180,E1 14113.368,E2 14113.368} C_VEL
LIN {X 0,Y 363.751,Z 666.373,A -85,B 0,C 180,E1 14119.204,E2 14119.204} C_VEL
LIN {X 0,Y 365.747,Z 667.451,A -85,B 0,C 180,E1 14124.953,E2 14124.953} C_VEL
LIN {X 0,Y 366.307,Z 668.34,A -85,B 0,C 180,E1 14130,E2 14130} C_VEL
LIN {X 0,Y 365.692,Z 666.854,A -85,B 0,C 180,E1 14135.642,E2 14135.642} C_VEL
LIN {X 0,Y 363.168,Z 666.113,A -85,B 0,C 180,E1 14142.032,E2 14142.032} C_VEL
LIN {X 0,Y 359.269,Z 663.294,A -85,B 0,C 180,E1 14148.108,E2 14148.108} C_VEL
LIN {X 0,Y 356.286,Z 658.492,A -85,B 0,C 180,E1 14152,E2 14152} C_VEL
LIN {X 0,Y 350.923,Z 654.651,A -85,B 0,C 180,E1 14157.3,E2 14157.3} C_VEL
LIN {X 0,Y 347.893,Z 650.244,A -85,B 0,C 180,E1 14160.133,E2 14160.133} C_VEL
LIN {X 0,Y 342.592,Z 645.198,A -85,B 0,C 180,E1 14164.405,E2 14164.405} C_VEL
LIN {X 0,Y 340.69,Z 642.453,A -85,B 0,C 180,E1 14165.922,E2 14165.922} C_VEL
LIN {X 0,Y 335.568,Z 637.483,A -85,B 0,C 180,E1 14169.598,E2 14169.598} C_VEL
LIN {X 0,Y 333.374,Z 634.431,A -85,B 0,C 180,E1 14171.177,E2 14171.177} C_VEL
LIN {X 0,Y 328.494,Z 629.333,A -85,B 0,C 180,E1 14174.421,E2 14174.421} C_VEL
LIN {X 0,Y 327.196,Z 627.004,A -85,B 0,C 180,E1 14175.332,E2 14175.332} C_VEL
LIN {X 0,Y 322.214,Z 622.256,A -85,B 0,C 180,E1 14178.432,E2 14178.432} C_VEL
LIN {X 0,Y 320.608,Z 619.335,A -85,B 0,C 180,E1 14179.505,E2 14179.505} C_VEL
LIN {X 0,Y 316.336,Z 615.465,A -85,B 0,C 180,E1 14181.969,E2 14181.969} C_VEL
LIN {X 0,Y 315.592,Z 611.91,A -85,B 0,C 180,E1 14182.76,E2 14182.76} C_VEL
LIN {X 0,Y 315.85,Z 611.91,A -85,B 0,C 180,E1 14191.352,E2 14191.352} C_VEL
LIN {X 0,Y 316.176,Z 611.91,A -85,B 0,C 180,E1 14197.47,E2 14197.47} C_VEL
LIN {X 0,Y 316.466,Z 611.91,A -85,B 0,C 180,E1 14203.314,E2 14203.314} C_VEL
LIN {X 0,Y 317.003,Z 611.91,A -85,B 0,C 180,E1 14211.757,E2 14211.757} C_VEL
LIN {X 0,Y 317.681,Z 611.91,A -85,B 0,C 180,E1 14219.995,E2 14219.995} C_VEL
LIN {X 0,Y 316.987,Z 611.91,A -85,B 0,C 180,E1 14228.233,E2 14228.233} C_VEL
LIN {X 0,Y 316.485,Z 611.91,A -85,B 0,C 180,E1 14236.675,E2 14236.675} C_VEL
LIN {X 0,Y 316.053,Z 611.91,A -85,B 0,C 180,E1 14244.468,E2 14244.468} C_VEL
LIN {X 0,Y 315.732,Z 611.91,A -85,B 0,C 180,E1 14251.829,E2 14251.829} C_VEL
LIN {X 0,Y 315.706,Z 611.91,A -85,B 0,C 180,E1 14254.733,E2 14254.733} C_VEL
LIN {X 0,Y 317.848,Z 617.32,A -85,B 0,C 180,E1 14255.518,E2 14255.518} C_VEL
LIN {X 0,Y 325.101,Z 627.796,A -85,B 0,C 180,E1 14257.63,E2 14257.63} C_VEL
LIN {X 0,Y 341.547,Z 655.023,A -85,B 0,C 180,E1 14262.096,E2 14262.096} C_VEL
LIN {X 0,Y 354.103,Z 683.416,A -85,B 0,C 180,E1 14265.919,E2 14265.919} C_VEL
LIN {X 0,Y 358.898,Z 699.691,A -85,B 0,C 180,E1 14267.886,E2 14267.886} C_VEL
LIN {X 0,Y 351.464,Z 735.541,A -85,B 0,C 180,E1 14270.502,E2 14270.502} C_VEL
LIN {X 0,Y 342.741,Z 768.839,A -85,B 0,C 180,E1 14274.175,E2 14274.175} C_VEL
LIN {X 0,Y 334.996,Z 795.462,A -85,B 0,C 180,E1 14278.304,E2 14278.304} C_VEL
LIN {X 0,Y 327.201,Z 821.235,A -85,B 0,C 180,E1 14283.946,E2 14283.946} C_VEL
LIN {X 0,Y 322.039,Z 839.982,A -85,B 0,C 180,E1 14289.816,E2 14289.816} C_VEL
LIN {X 0,Y 319.073,Z 854.03,A -85,B 0,C 180,E1 14296.275,E2 14296.275} C_VEL
LIN {X 0,Y 318.118,Z 861.517,A -85,B 0,C 180,E1 14301.791,E2 14301.791} C_VEL
LIN {X 0,Y 317.874,Z 865.181,A -85,B 0,C 180,E1 14307.27,E2 14307.27} C_VEL
LIN {X 0,Y 317.901,Z 865.182,A -85,B 0,C 180,E1 14312.73,E2 14312.73} C_VEL
LIN {X 0,Y 318.115,Z 861.517,A -85,B 0,C 180,E1 14318.209,E2 14318.209} C_VEL
LIN {X 0,Y 319.253,Z 852.758,A -85,B 0,C 180,E1 14324.417,E2 14324.417} C_VEL
LIN {X 0,Y 322.415,Z 838.432,A -85,B 0,C 180,E1 14330.783,E2 14330.783} C_VEL
LIN {X 0,Y 328.195,Z 817.668,A -85,B 0,C 180,E1 14336.956,E2 14336.956} C_VEL
LIN {X 0,Y 335.689,Z 792.989,A -85,B 0,C 180,E1 14342.136,E2 14342.136} C_VEL
LIN {X 0,Y 344.494,Z 762.862,A -85,B 0,C 180,E1 14346.589,E2 14346.589} C_VEL
LIN {X 0,Y 349.16,Z 744.852,A -85,B 0,C 180,E1 14348.597,E2 14348.597} C_VEL
LIN {X 0,Y 349.419,Z 718.057,A -85,B 0,C 180,E1 14351.732,E2 14351.732} C_VEL
LIN {X 0,Y 349.756,Z 716.108,A -85,B 0,C 180,E1 14351.883,E2 14351.883} C_VEL
LIN {X 0,Y 352.226,Z 699.911,A -85,B 0,C 180,E1 14353.06,E2 14353.06} C_VEL
LIN {X 0,Y 341.538,Z 670.216,A -85,B 0,C 180,E1 14357.041,E2 14357.041} C_VEL
LIN {X 0,Y 326.811,Z 642.196,A -85,B 0,C 180,E1 14361.437,E2 14361.437} C_VEL
LIN {X 0,Y 310.838,Z 618.074,A -85,B 0,C 180,E1 14366.289,E2 14366.289} C_VEL
LIN {X 0,Y 307.994,Z 613.553,A -85,B 0,C 180,E1 14367.273,E2 14367.273} C_VEL
LIN {X 0,Y 307.842,Z 611.91,A -85,B 0,C 180,E1 14367.64,E2 14367.64} C_VEL
LIN {X 0,Y 307.99,Z 611.91,A -85,B 0,C 180,E1 14373.748,E2 14373.748} C_VEL
LIN {X 0,Y 308.314,Z 611.91,A -85,B 0,C 180,E1 14379.901,E2 14379.901} C_VEL
LIN {X 0,Y 308.682,Z 611.91,A -85,B 0,C 180,E1 14385.81,E2 14385.81} C_VEL
LIN {X 0,Y 309.285,Z 611.91,A -85,B 0,C 180,E1 14394.387,E2 14394.387} C_VEL
LIN {X 0,Y 309.711,Z 611.91,A -85,B 0,C 180,E1 14400.005,E2 14400.005} C_VEL
LIN {X 0,Y 309.303,Z 611.91,A -85,B 0,C 180,E1 14405.623,E2 14405.623} C_VEL
LIN {X 0,Y 308.668,Z 611.91,A -85,B 0,C 180,E1 14414.202,E2 14414.202} C_VEL
LIN {X 0,Y 308.222,Z 611.91,A -85,B 0,C 180,E1 14421.041,E2 14421.041} C_VEL
LIN {X 0,Y 307.873,Z 611.91,A -85,B 0,C 180,E1 14429.462,E2 14429.462} C_VEL
LIN {X 0,Y 307.656,Z 611.91,A -85,B 0,C 180,E1 14433.877,E2 14433.877} C_VEL
LIN {X 0,Y 309.318,Z 616.682,A -85,B 0,C 180,E1 14434.881,E2 14434.881} C_VEL
LIN {X 0,Y 313.58,Z 620.682,A -85,B 0,C 180,E1 14437.066,E2 14437.066} C_VEL
LIN {X 0,Y 317.357,Z 625.986,A -85,B 0,C 180,E1 14439.258,E2 14439.258} C_VEL
LIN {X 0,Y 320.175,Z 628.67,A -85,B 0,C 180,E1 14440.912,E2 14440.912} C_VEL
LIN {X 0,Y 324.895,Z 634.117,A -85,B 0,C 180,E1 14443.898,E2 14443.898} C_VEL
LIN {X 0,Y 331.322,Z 641.733,A -85,B 0,C 180,E1 14448.158,E2 14448.158} C_VEL
LIN {X 0,Y 334.003,Z 644.922,A -85,B 0,C 180,E1 14450.006,E2 14450.006} C_VEL
LIN {X 0,Y 339.19,Z 650.08,A -85,B 0,C 180,E1 14453.73,E2 14453.73} C_VEL
LIN {X 0,Y 344.82,Z 656.926,A -85,B 0,C 180,E1 14458.204,E2 14458.204} C_VEL
LIN {X 0,Y 348.211,Z 659.918,A -85,B 0,C 180,E1 14461.042,E2 14461.042} C_VEL
LIN {X 0,Y 352.4,Z 664.879,A -85,B 0,C 180,E1 14465.082,E2 14465.082} C_VEL
LIN {X 0,Y 356.046,Z 667.672,A -85,B 0,C 180,E1 14468.945,E2 14468.945} C_VEL
LIN {X 0,Y 359.534,Z 672.417,A -85,B 0,C 180,E1 14473.67,E2 14473.67} C_VEL
LIN {X 0,Y 362.586,Z 674.136,A -85,B 0,C 180,E1 14478.821,E2 14478.821} C_VEL
LIN {X 0,Y 364.732,Z 675.156,A -85,B 0,C 180,E1 14484.661,E2 14484.661} C_VEL
LIN {X 0,Y 365.346,Z 676.168,A -85,B 0,C 180,E1 14490,E2 14490} C_VEL
LIN {X 0,Y 364.719,Z 674.741,A -85,B 0,C 180,E1 14495.657,E2 14495.657} C_VEL
LIN {X 0,Y 362.187,Z 673.949,A -85,B 0,C 180,E1 14502.065,E2 14502.065} C_VEL
LIN {X 0,Y 358.289,Z 671.169,A -85,B 0,C 180,E1 14508.108,E2 14508.108} C_VEL
LIN {X 0,Y 354.708,Z 666.137,A -85,B 0,C 180,E1 14512.592,E2 14512.592} C_VEL
LIN {X 0,Y 349.433,Z 662.012,A -85,B 0,C 180,E1 14517.743,E2 14517.743} C_VEL
LIN {X 0,Y 346.486,Z 657.879,A -85,B 0,C 180,E1 14520.493,E2 14520.493} C_VEL
LIN {X 0,Y 341.132,Z 652.689,A -85,B 0,C 180,E1 14524.753,E2 14524.753} C_VEL
LIN {X 0,Y 338.913,Z 649.913,A -85,B 0,C 180,E1 14526.469,E2 14526.469} C_VEL
LIN {X 0,Y 333.696,Z 644.341,A -85,B 0,C 180,E1 14530.218,E2 14530.218} C_VEL
LIN {X 0,Y 330.712,Z 641.339,A -85,B 0,C 180,E1 14532.23,E2 14532.23} C_VEL
LIN {X 0,Y 326.244,Z 635.448,A -85,B 0,C 180,E1 14535.256,E2 14535.256} C_VEL
LIN {X 0,Y 320.214,Z 629.121,A -85,B 0,C 180,E1 14539.036,E2 14539.036} C_VEL
LIN {X 0,Y 318.145,Z 626.554,A -85,B 0,C 180,E1 14540.309,E2 14540.309} C_VEL
LIN {X 0,Y 313.853,Z 621.666,A -85,B 0,C 180,E1 14542.74,E2 14542.74} C_VEL
LIN {X 0,Y 312.632,Z 619.247,A -85,B 0,C 180,E1 14543.492,E2 14543.492} C_VEL
LIN {X 0,Y 308.198,Z 614.867,A -85,B 0,C 180,E1 14545.724,E2 14545.724} C_VEL
LIN {X 0,Y 307.612,Z 611.91,A -85,B 0,C 180,E1 14546.322,E2 14546.322} C_VEL
LIN {X 0,Y 308.014,Z 611.91,A -85,B 0,C 180,E1 14553.738,E2 14553.738} C_VEL
LIN {X 0,Y 308.368,Z 611.91,A -85,B 0,C 180,E1 14559.893,E2 14559.893} C_VEL
LIN {X 0,Y 308.616,Z 611.91,A -85,B 0,C 180,E1 14565.796,E2 14565.796} C_VEL
LIN {X 0,Y 309.298,Z 611.91,A -85,B 0,C 180,E1 14574.377,E2 14574.377} C_VEL
LIN {X 0,Y 309.776,Z 611.91,A -85,B 0,C 180,E1 14579.995,E2 14579.995} C_VEL
LIN {X 0,Y 309.046,Z 611.91,A -85,B 0,C 180,E1 14588.446,E2 14588.446} C_VEL
LIN {X 0,Y 308.686,Z 611.91,A -85,B 0,C 180,E1 14594.19,E2 14594.19} C_VEL
LIN {X 0,Y 308.236,Z 611.91,A -85,B 0,C 180,E1 14601.048,E2 14601.048} C_VEL
LIN {X 0,Y 307.874,Z 611.91,A -85,B 0,C 180,E1 14609.45,E2 14609.45} C_VEL
LIN {X 0,Y 307.841,Z 612.729,A -85,B 0,C 180,E1 14612.648,E2 14612.648} C_VEL
LIN {X 0,Y 310.591,Z 617.942,A -85,B 0,C 180,E1 14613.638,E2 14613.638} C_VEL
LIN {X 0,Y 324.15,Z 637.95,A -85,B 0,C 180,E1 14617.793,E2 14617.793} C_VEL
LIN {X 0,Y 339.767,Z 666.155,A -85,B 0,C 180,E1 14622.368,E2 14622.368} C_VEL
LIN {X 0,Y 350.967,Z 695.432,A -85,B 0,C 180,E1 14626.352,E2 14626.352} C_VEL
LIN {X 0,Y 352.375,Z 702.933,A -85,B 0,C 180,E1 14627.23,E2 14627.23} C_VEL
LIN {X 0,Y 344.776,Z 737.453,A -85,B 0,C 180,E1 14629.862,E2 14629.862} C_VEL
LIN {X 0,Y 335.567,Z 770.993,A -85,B 0,C 180,E1 14633.687,E2 14633.687} C_VEL
LIN {X 0,Y 327.02,Z 798.603,A -85,B 0,C 180,E1 14638.221,E2 14638.221} C_VEL
LIN {X 0,Y 319.588,Z 822.246,A -85,B 0,C 180,E1 14643.633,E2 14643.633} C_VEL
LIN {X 0,Y 313.812,Z 842.16,A -85,B 0,C 180,E1 14650.261,E2 14650.261} C_VEL
LIN {X 0,Y 311.021,Z 855.147,A -85,B 0,C 180,E1 14656.774,E2 14656.774} C_VEL
LIN {X 0,Y 310.124,Z 862.456,A -85,B 0,C 180,E1 14662.989,E2 14662.989} C_VEL
LIN {X 0,Y 309.97,Z 864.947,A -85,B 0,C 180,E1 14667.2,E2 14667.2} C_VEL
LIN {X 0,Y 309.997,Z 864.948,A -85,B 0,C 180,E1 14672.8,E2 14672.8} C_VEL
LIN {X 0,Y 310.227,Z 861.281,A -85,B 0,C 180,E1 14678.419,E2 14678.419} C_VEL
LIN {X 0,Y 311.486,Z 852.521,A -85,B 0,C 180,E1 14684.785,E2 14684.785} C_VEL
LIN {X 0,Y 314.731,Z 838.591,A -85,B 0,C 180,E1 14691.149,E2 14691.149} C_VEL
LIN {X 0,Y 320.317,Z 819.579,A -85,B 0,C 180,E1 14697.06,E2 14697.06} C_VEL
LIN {X 0,Y 328.086,Z 795.221,A -85,B 0,C 180,E1 14702.444,E2 14702.444} C_VEL
LIN {X 0,Y 337.012,Z 766.212,A -85,B 0,C 180,E1 14706.933,E2 14706.933} C_VEL
LIN {X 0,Y 345.525,Z 734.329,A -85,B 0,C 180,E1 14710.431,E2 14710.431} C_VEL
LIN {X 0,Y 349.756,Z 716.108,A -85,B 0,C 180,E1 14711.883,E2 14711.883} C_VEL
LIN {X 0,Y 348.986,Z 707.825,A -85,B 0,C 180,E1 14712.837,E2 14712.837} C_VEL
LIN {X 0,Y 344.767,Z 698.373,A -85,B 0,C 180,E1 14714.343,E2 14714.343} C_VEL
LIN {X 0,Y 333.768,Z 668.993,A -85,B 0,C 180,E1 14718.555,E2 14718.555} C_VEL
LIN {X 0,Y 319.054,Z 641.959,A -85,B 0,C 180,E1 14723.214,E2 14723.214} C_VEL
LIN {X 0,Y 306.729,Z 623.662,A -85,B 0,C 180,E1 14727.212,E2 14727.212} C_VEL
LIN {X 0,Y 302.96,Z 618.103,A -85,B 0,C 180,E1 14728.572,E2 14728.572} C_VEL
LIN {X 0,Y 300.066,Z 613.231,A -85,B 0,C 180,E1 14729.704,E2 14729.704} C_VEL
LIN {X 0,Y 299.959,Z 611.91,A -85,B 0,C 180,E1 14729.915,E2 14729.915} C_VEL
LIN {X 0,Y 300.122,Z 611.91,A -85,B 0,C 180,E1 14736.204,E2 14736.204} C_VEL
LIN {X 0,Y 300.634,Z 611.91,A -85,B 0,C 180,E1 14743.113,E2 14743.113} C_VEL
LIN {X 0,Y 301.118,Z 611.91,A -85,B 0,C 180,E1 14751.33,E2 14751.33} C_VEL
LIN {X 0,Y 301.648,Z 611.91,A -85,B 0,C 180,E1 14757.128,E2 14757.128} C_VEL
LIN {X 0,Y 301.694,Z 611.91,A -85,B 0,C 180,E1 14762.882,E2 14762.882} C_VEL
LIN {X 0,Y 300.922,Z 611.91,A -85,B 0,C 180,E1 14771.615,E2 14771.615} C_VEL
LIN {X 0,Y 300.557,Z 611.91,A -85,B 0,C 180,E1 14777.598,E2 14777.598} C_VEL
LIN {X 0,Y 300.079,Z 611.91,A -85,B 0,C 180,E1 14784.743,E2 14784.743} C_VEL
LIN {X 0,Y 299.792,Z 611.991,A -85,B 0,C 180,E1 14790.732,E2 14790.732} C_VEL
LIN {X 0,Y 301.623,Z 617.024,A -85,B 0,C 180,E1 14791.729,E2 14791.729} C_VEL
LIN {X 0,Y 305.291,Z 620.459,A -85,B 0,C 180,E1 14793.402,E2 14793.402} C_VEL
LIN {X 0,Y 309.666,Z 626.093,A -85,B 0,C 180,E1 14795.605,E2 14795.605} C_VEL
LIN {X 0,Y 312.005,Z 628.965,A -85,B 0,C 180,E1 14796.825,E2 14796.825} C_VEL
LIN {X 0,Y 316.899,Z 634.255,A -85,B 0,C 180,E1 14799.578,E2 14799.578} C_VEL
LIN {X 0,Y 323.282,Z 641.652,A -85,B 0,C 180,E1 14803.529,E2 14803.529} C_VEL
LIN {X 0,Y 329.939,Z 649.368,A -85,B 0,C 180,E1 14807.922,E2 14807.922} C_VEL
LIN {X 0,Y 337.126,Z 657.396,A -85,B 0,C 180,E1 14812.97,E2 14812.97} C_VEL
LIN {X 0,Y 339.843,Z 660.6,A -85,B 0,C 180,E1 14815.046,E2 14815.046} C_VEL
LIN {X 0,Y 345.432,Z 665.753,A -85,B 0,C 180,E1 14819.463,E2 14819.463} C_VEL
LIN {X 0,Y 351.007,Z 672.431,A -85,B 0,C 180,E1 14824.659,E2 14824.659} C_VEL
LIN {X 0,Y 354.956,Z 675.511,A -85,B 0,C 180,E1 14828.815,E2 14828.815} C_VEL
LIN {X 0,Y 358.374,Z 680.138,A -85,B 0,C 180,E1 14833.431,E2 14833.431} C_VEL
LIN {X 0,Y 361.922,Z 682.048,A -85,B 0,C 180,E1 14839.393,E2 14839.393} C_VEL
LIN {X 0,Y 363.817,Z 683.166,A -85,B 0,C 180,E1 14844.968,E2 14844.968} C_VEL
LIN {X 0,Y 364.386,Z 683.986,A -85,B 0,C 180,E1 14850,E2 14850} C_VEL
LIN {X 0,Y 363.736,Z 682.502,A -85,B 0,C 180,E1 14855.823,E2 14855.823} C_VEL
LIN {X 0,Y 361.205,Z 681.784,A -85,B 0,C 180,E1 14862.098,E2 14862.098} C_VEL
LIN {X 0,Y 357.266,Z 678.985,A -85,B 0,C 180,E1 14868.162,E2 14868.162} C_VEL
LIN {X 0,Y 353.663,Z 673.959,A -85,B 0,C 180,E1 14872.662,E2 14872.662} C_VEL
LIN {X 0,Y 348.33,Z 669.859,A -85,B 0,C 180,E1 14877.838,E2 14877.838} C_VEL
LIN {X 0,Y 345.012,Z 665.499,A -85,B 0,C 180,E1 14880.856,E2 14880.856} C_VEL
LIN {X 0,Y 339.618,Z 660.03,A -85,B 0,C 180,E1 14885.165,E2 14885.165} C_VEL
LIN {X 0,Y 336.664,Z 657.033,A -85,B 0,C 180,E1 14887.344,E2 14887.344} C_VEL
LIN {X 0,Y 331.416,Z 650.435,A -85,B 0,C 180,E1 14891.126,E2 14891.126} C_VEL
LIN {X 0,Y 325.358,Z 644.42,A -85,B 0,C 180,E1 14895.101,E2 14895.101} C_VEL
LIN {X 0,Y 322.57,Z 641.325,A -85,B 0,C 180,E1 14896.881,E2 14896.881} C_VEL
LIN {X 0,Y 317.734,Z 635.022,A -85,B 0,C 180,E1 14899.937,E2 14899.937} C_VEL
LIN {X 0,Y 312.092,Z 629.352,A -85,B 0,C 180,E1 14903.107,E2 14903.107} C_VEL
LIN {X 0,Y 309.655,Z 626.179,A -85,B 0,C 180,E1 14904.393,E2 14904.393} C_VEL
LIN {X 0,Y 305.26,Z 620.536,A -85,B 0,C 180,E1 14906.607,E2 14906.607} C_VEL
LIN {X 0,Y 300.101,Z 614.248,A -85,B 0,C 180,E1 14909.024,E2 14909.024} C_VEL
LIN {X 0,Y 299.789,Z 611.91,A -85,B 0,C 180,E1 14909.469,E2 14909.469} C_VEL
LIN {X 0,Y 300.19,Z 611.91,A -85,B 0,C 180,E1 14916.199,E2 14916.199} C_VEL
LIN {X 0,Y 300.637,Z 611.91,A -85,B 0,C 180,E1 14923.111,E2 14923.111} C_VEL
LIN {X 0,Y 301.104,Z 611.91,A -85,B 0,C 180,E1 14931.748,E2 14931.748} C_VEL
LIN {X 0,Y 301.884,Z 611.91,A -85,B 0,C 180,E1 14939.995,E2 14939.995} C_VEL
LIN {X 0,Y 301.118,Z 611.91,A -85,B 0,C 180,E1 14948.67,E2 14948.67} C_VEL
LIN {X 0,Y 300.642,Z 611.91,A -85,B 0,C 180,E1 14956.893,E2 14956.893} C_VEL
LIN {X 0,Y 300.088,Z 611.91,A -85,B 0,C 180,E1 14964.747,E2 14964.747} C_VEL
LIN {X 0,Y 299.948,Z 611.932,A -85,B 0,C 180,E1 14970.197,E2 14970.197} C_VEL
LIN {X 0,Y 301.97,Z 617.206,A -85,B 0,C 180,E1 14971.082,E2 14971.082} C_VEL
LIN {X 0,Y 304.843,Z 620.598,A -85,B 0,C 180,E1 14972.106,E2 14972.106} C_VEL
LIN {X 0,Y 320.411,Z 644.107,A -85,B 0,C 180,E1 14977.207,E2 14977.207} C_VEL
LIN {X 0,Y 334.854,Z 671.439,A -85,B 0,C 180,E1 14981.822,E2 14981.822} C_VEL
LIN {X 0,Y 345.306,Z 700.358,A -85,B 0,C 180,E1 14985.925,E2 14985.925} C_VEL
LIN {X 0,Y 346.077,Z 705.235,A -85,B 0,C 180,E1 14986.49,E2 14986.49} C_VEL
LIN {X 0,Y 338.425,Z 738.224,A -85,B 0,C 180,E1 14989.089,E2 14989.089} C_VEL
LIN {X 0,Y 328.756,Z 771.948,A -85,B 0,C 180,E1 14993.017,E2 14993.017} C_VEL
LIN {X 0,Y 319.606,Z 800.054,A -85,B 0,C 180,E1 14997.796,E2 14997.796} C_VEL
LIN {X 0,Y 311.924,Z 823.213,A -85,B 0,C 180,E1 15003.321,E2 15003.321} C_VEL
LIN {X 0,Y 306.021,Z 842.626,A -85,B 0,C 180,E1 15010.036,E2 15010.036} C_VEL
LIN {X 0,Y 303.135,Z 855.288,A -85,B 0,C 180,E1 15016.694,E2 15016.694} C_VEL
LIN {X 0,Y 302.238,Z 862.221,A -85,B 0,C 180,E1 15022.806,E2 15022.806} C_VEL
LIN {X 0,Y 302.066,Z 864.713,A -85,B 0,C 180,E1 15027.127,E2 15027.127} C_VEL
LIN {X 0,Y 302.092,Z 864.714,A -85,B 0,C 180,E1 15032.873,E2 15032.873} C_VEL
LIN {X 0,Y 302.341,Z 861.045,A -85,B 0,C 180,E1 15038.64,E2 15038.64} C_VEL
LIN {X 0,Y 303.715,Z 852.284,A -85,B 0,C 180,E1 15045.172,E2 15045.172} C_VEL
LIN {X 0,Y 307.208,Z 838.352,A -85,B 0,C 180,E1 15051.693,E2 15051.693} C_VEL
LIN {X 0,Y 313.125,Z 819.335,A -85,B 0,C 180,E1 15057.736,E2 15057.736} C_VEL
LIN {X 0,Y 321.291,Z 794.982,A -85,B 0,C 180,E1 15063.217,E2 15063.217} C_VEL
LIN {X 0,Y 330.63,Z 765.975,A -85,B 0,C 180,E1 15067.769,E2 15067.769} C_VEL
LIN {X 0,Y 339.427,Z 734.336,A -85,B 0,C 180,E1 15071.284,E2 15071.284} C_VEL
LIN {X 0,Y 346.132,Z 703.456,A -85,B 0,C 180,E1 15073.663,E2 15073.663} C_VEL
LIN {X 0,Y 344.767,Z 698.373,A -85,B 0,C 180,E1 15074.343,E2 15074.343} C_VEL
LIN {X 0,Y 340.071,Z 690.159,A -85,B 0,C 180,E1 15075.866,E2 15075.866} C_VEL
LIN {X 0,Y 330.445,Z 677.925,A -85,B 0,C 180,E1 15078.563,E2 15078.563} C_VEL
LIN {X 0,Y 317.926,Z 652.608,A -85,B 0,C 180,E1 15082.942,E2 15082.942} C_VEL
LIN {X 0,Y 304.224,Z 630.852,A -85,B 0,C 180,E1 15087.635,E2 15087.635} C_VEL
LIN {X 0,Y 295.618,Z 618.498,A -85,B 0,C 180,E1 15090.944,E2 15090.944} C_VEL
LIN {X 0,Y 292.304,Z 613.744,A -85,B 0,C 180,E1 15092.369,E2 15092.369} C_VEL
LIN {X 0,Y 292.137,Z 611.91,A -85,B 0,C 180,E1 15092.794,E2 15092.794} C_VEL
LIN {X 0,Y 292.545,Z 611.91,A -85,B 0,C 180,E1 15101.915,E2 15101.915} C_VEL
LIN {X 0,Y 293.025,Z 611.91,A -85,B 0,C 180,E1 15109.03,E2 15109.03} C_VEL
LIN {X 0,Y 293.723,Z 611.91,A -85,B 0,C 180,E1 15117.051,E2 15117.051} C_VEL
LIN {X 0,Y 293.768,Z 611.91,A -85,B 0,C 180,E1 15122.96,E2 15122.96} C_VEL
LIN {X 0,Y 292.986,Z 611.91,A -85,B 0,C 180,E1 15131.934,E2 15131.934} C_VEL
LIN {X 0,Y 292.565,Z 611.91,A -85,B 0,C 180,E1 15138.095,E2 15138.095} C_VEL
LIN {X 0,Y 292.193,Z 611.91,A -85,B 0,C 180,E1 15144.495,E2 15144.495} C_VEL
LIN {X 0,Y 292.027,Z 611.91,A -85,B 0,C 180,E1 15147.82,E2 15147.82} C_VEL
LIN {X 0,Y 293.837,Z 617.086,A -85,B 0,C 180,E1 15148.779,E2 15148.779} C_VEL
LIN {X 0,Y 297.262,Z 620.517,A -85,B 0,C 180,E1 15150.229,E2 15150.229} C_VEL
LIN {X 0,Y 301.667,Z 626.087,A -85,B 0,C 180,E1 15152.231,E2 15152.231} C_VEL
LIN {X 0,Y 308.077,Z 633.747,A -85,B 0,C 180,E1 15155.384,E2 15155.384} C_VEL
LIN {X 0,Y 314.433,Z 641.384,A -85,B 0,C 180,E1 15158.901,E2 15158.901} C_VEL
LIN {X 0,Y 321.923,Z 649.365,A -85,B 0,C 180,E1 15163.374,E2 15163.374} C_VEL
LIN {X 0,Y 328.312,Z 656.885,A -85,B 0,C 180,E1 15167.554,E2 15167.554} C_VEL
LIN {X 0,Y 335.662,Z 664.958,A -85,B 0,C 180,E1 15172.665,E2 15172.665} C_VEL
LIN {X 0,Y 338.688,Z 668.552,A -85,B 0,C 180,E1 15174.945,E2 15174.945} C_VEL
LIN {X 0,Y 345.754,Z 675.538,A -85,B 0,C 180,E1 15180.692,E2 15180.692} C_VEL
LIN {X 0,Y 350.479,Z 680.621,A -85,B 0,C 180,E1 15185.126,E2 15185.126} C_VEL
LIN {X 0,Y 353.831,Z 683.32,A -85,B 0,C 180,E1 15188.644,E2 15188.644} C_VEL
LIN {X 0,Y 357.6,Z 688.141,A -85,B 0,C 180,E1 15193.71,E2 15193.71} C_VEL
LIN {X 0,Y 360.938,Z 689.884,A -85,B 0,C 180,E1 15199.363,E2 15199.363} C_VEL
LIN {X 0,Y 362.84,Z 690.998,A -85,B 0,C 180,E1 15204.913,E2 15204.913} C_VEL
LIN {X 0,Y 363.391,Z 691.793,A -85,B 0,C 180,E1 15210.322,E2 15210.322} C_VEL
LIN {X 0,Y 362.753,Z 690.288,A -85,B 0,C 180,E1 15215.989,E2 15215.989} C_VEL
LIN {X 0,Y 360.218,Z 689.611,A -85,B 0,C 180,E1 15222.132,E2 15222.132} C_VEL
LIN {X 0,Y 356.236,Z 686.809,A -85,B 0,C 180,E1 15228.216,E2 15228.216} C_VEL
LIN {X 0,Y 352.309,Z 681.68,A -85,B 0,C 180,E1 15233.056,E2 15233.056} C_VEL
LIN {X 0,Y 346.706,Z 676.996,A -85,B 0,C 180,E1 15238.441,E2 15238.441} C_VEL
LIN {X 0,Y 343.446,Z 673.048,A -85,B 0,C 180,E1 15241.292,E2 15241.292} C_VEL
LIN {X 0,Y 338.054,Z 667.353,A -85,B 0,C 180,E1 15245.581,E2 15245.581} C_VEL
LIN {X 0,Y 330.804,Z 659.655,A -85,B 0,C 180,E1 15250.774,E2 15250.774} C_VEL
LIN {X 0,Y 323.284,Z 651.186,A -85,B 0,C 180,E1 15255.741,E2 15255.741} C_VEL
LIN {X 0,Y 316.212,Z 643.225,A -85,B 0,C 180,E1 15260.075,E2 15260.075} C_VEL
LIN {X 0,Y 309.696,Z 636.075,A -85,B 0,C 180,E1 15263.73,E2 15263.73} C_VEL
LIN {X 0,Y 302.939,Z 627.56,A -85,B 0,C 180,E1 15267.178,E2 15267.178} C_VEL
LIN {X 0,Y 297.429,Z 620.919,A -85,B 0,C 180,E1 15269.691,E2 15269.691} C_VEL
LIN {X 0,Y 295.311,Z 618.423,A -85,B 0,C 180,E1 15270.594,E2 15270.594} C_VEL
LIN {X 0,Y 292.228,Z 613.825,A -85,B 0,C 180,E1 15271.977,E2 15271.977} C_VEL
LIN {X 0,Y 292.033,Z 611.91,A -85,B 0,C 180,E1 15272.181,E2 15272.181} C_VEL
LIN {X 0,Y 292.421,Z 611.91,A -85,B 0,C 180,E1 15278.745,E2 15278.745} C_VEL
LIN {X 0,Y 292.747,Z 611.91,A -85,B 0,C 180,E1 15285.008,E2 15285.008} C_VEL
LIN {X 0,Y 293.432,Z 611.91,A -85,B 0,C 180,E1 15294.072,E2 15294.072} C_VEL
LIN {X 0,Y 293.978,Z 611.91,A -85,B 0,C 180,E1 15299.995,E2 15299.995} C_VEL
LIN {X 0,Y 293.442,Z 611.91,A -85,B 0,C 180,E1 15305.917,E2 15305.917} C_VEL
LIN {X 0,Y 293.008,Z 611.91,A -85,B 0,C 180,E1 15311.923,E2 15311.923} C_VEL
LIN {X 0,Y 292.563,Z 611.91,A -85,B 0,C 180,E1 15318.083,E2 15318.083} C_VEL
LIN {X 0,Y 292.135,Z 611.91,A -85,B 0,C 180,E1 15327.21,E2 15327.21} C_VEL
LIN {X 0,Y 294.64,Z 617.754,A -85,B 0,C 180,E1 15328.678,E2 15328.678} C_VEL
LIN {X 0,Y 297.116,Z 620.462,A -85,B 0,C 180,E1 15329.661,E2 15329.661} C_VEL
LIN {X 0,Y 311.416,Z 641.849,A -85,B 0,C 180,E1 15334.881,E2 15334.881} C_VEL
LIN {X 0,Y 325.714,Z 667.378,A -85,B 0,C 180,E1 15339.721,E2 15339.721} C_VEL
LIN {X 0,Y 336.658,Z 694.836,A -85,B 0,C 180,E1 15343.981,E2 15343.981} C_VEL
LIN {X 0,Y 339.829,Z 707.573,A -85,B 0,C 180,E1 15345.726,E2 15345.726} C_VEL
LIN {X 0,Y 331.272,Z 742.209,A -85,B 0,C 180,E1 15348.613,E2 15348.613} C_VEL
LIN {X 0,Y 321.996,Z 772.825,A -85,B 0,C 180,E1 15352.318,E2 15352.318} C_VEL
LIN {X 0,Y 312.212,Z 801.505,A -85,B 0,C 180,E1 15357.35,E2 15357.35} C_VEL
LIN {X 0,Y 304.276,Z 824.15,A -85,B 0,C 180,E1 15362.996,E2 15362.996} C_VEL
LIN {X 0,Y 298.271,Z 842.957,A -85,B 0,C 180,E1 15369.742,E2 15369.742} C_VEL
LIN {X 0,Y 295.372,Z 854.913,A -85,B 0,C 180,E1 15376.236,E2 15376.236} C_VEL
LIN {X 0,Y 294.365,Z 861.986,A -85,B 0,C 180,E1 15382.612,E2 15382.612} C_VEL
LIN {X 0,Y 294.162,Z 864.479,A -85,B 0,C 180,E1 15387.05,E2 15387.05} C_VEL
LIN {X 0,Y 294.186,Z 864.48,A -85,B 0,C 180,E1 15392.95,E2 15392.95} C_VEL
LIN {X 0,Y 294.46,Z 860.81,A -85,B 0,C 180,E1 15398.874,E2 15398.874} C_VEL
LIN {X 0,Y 295.939,Z 852.045,A -85,B 0,C 180,E1 15405.581,E2 15405.581} C_VEL
LIN {X 0,Y 299.707,Z 838.113,A -85,B 0,C 180,E1 15412.265,E2 15412.265} C_VEL
LIN {X 0,Y 305.964,Z 819.096,A -85,B 0,C 180,E1 15418.443,E2 15418.443} C_VEL
LIN {X 0,Y 314.556,Z 794.743,A -85,B 0,C 180,E1 15424.024,E2 15424.024} C_VEL
LIN {X 0,Y 324.288,Z 765.736,A -85,B 0,C 180,E1 15428.643,E2 15428.643} C_VEL
LIN {X 0,Y 333.33,Z 734.594,A -85,B 0,C 180,E1 15432.148,E2 15432.148} C_VEL
LIN {X 0,Y 339.938,Z 707.31,A -85,B 0,C 180,E1 15434.281,E2 15434.281} C_VEL
LIN {X 0,Y 331.507,Z 680.383,A -85,B 0,C 180,E1 15438.174,E2 15438.174} C_VEL
LIN {X 0,Y 330.445,Z 677.925,A -85,B 0,C 180,E1 15438.563,E2 15438.563} C_VEL
LIN {X 0,Y 322.668,Z 668.871,A -85,B 0,C 180,E1 15440.823,E2 15440.823} C_VEL
LIN {X 0,Y 314.817,Z 660.163,A -85,B 0,C 180,E1 15443.203,E2 15443.203} C_VEL
LIN {X 0,Y 301.061,Z 637.263,A -85,B 0,C 180,E1 15448.279,E2 15448.279} C_VEL
LIN {X 0,Y 292.222,Z 624.803,A -85,B 0,C 180,E1 15451.834,E2 15451.834} C_VEL
LIN {X 0,Y 287.972,Z 618.641,A -85,B 0,C 180,E1 15453.778,E2 15453.778} C_VEL
LIN {X 0,Y 284.609,Z 614.152,A -85,B 0,C 180,E1 15455.437,E2 15455.437} C_VEL
LIN {X 0,Y 284.253,Z 611.91,A -85,B 0,C 180,E1 15455.836,E2 15455.836} C_VEL
LIN {X 0,Y 284.8,Z 611.91,A -85,B 0,C 180,E1 15464.591,E2 15464.591} C_VEL
LIN {X 0,Y 285.235,Z 611.91,A -85,B 0,C 180,E1 15470.843,E2 15470.843} C_VEL
LIN {X 0,Y 285.821,Z 611.91,A -85,B 0,C 180,E1 15476.969,E2 15476.969} C_VEL
LIN {X 0,Y 285.86,Z 611.91,A -85,B 0,C 180,E1 15483.041,E2 15483.041} C_VEL
LIN {X 0,Y 285.019,Z 611.91,A -85,B 0,C 180,E1 15492.273,E2 15492.273} C_VEL
LIN {X 0,Y 284.582,Z 611.91,A -85,B 0,C 180,E1 15498.621,E2 15498.621} C_VEL
LIN {X 0,Y 284.276,Z 612.56,A -85,B 0,C 180,E1 15504.738,E2 15504.738} C_VEL
LIN {X 0,Y 286.463,Z 617.546,A -85,B 0,C 180,E1 15505.963,E2 15505.963} C_VEL
LIN {X 0,Y 289.368,Z 620.419,A -85,B 0,C 180,E1 15507.284,E2 15507.284} C_VEL
LIN {X 0,Y 293.732,Z 626.089,A -85,B 0,C 180,E1 15509.217,E2 15509.217} C_VEL
LIN {X 0,Y 299.366,Z 633.353,A -85,B 0,C 180,E1 15511.761,E2 15511.761} C_VEL
LIN {X 0,Y 306.289,Z 641.387,A -85,B 0,C 180,E1 15515.188,E2 15515.188} C_VEL
LIN {X 0,Y 312.41,Z 648.828,A -85,B 0,C 180,E1 15518.579,E2 15518.579} C_VEL
LIN {X 0,Y 320.194,Z 656.955,A -85,B 0,C 180,E1 15523.15,E2 15523.15} C_VEL
LIN {X 0,Y 326.65,Z 664.46,A -85,B 0,C 180,E1 15527.305,E2 15527.305} C_VEL
LIN {X 0,Y 334.246,Z 672.728,A -85,B 0,C 180,E1 15532.559,E2 15532.559} C_VEL
LIN {X 0,Y 341.25,Z 680.247,A -85,B 0,C 180,E1 15537.95,E2 15537.95} C_VEL
LIN {X 0,Y 344.54,Z 683.632,A -85,B 0,C 180,E1 15540.692,E2 15540.692} C_VEL
LIN {X 0,Y 349.724,Z 688.755,A -85,B 0,C 180,E1 15545.56,E2 15545.56} C_VEL
LIN {X 0,Y 352.488,Z 691.132,A -85,B 0,C 180,E1 15548.503,E2 15548.503} C_VEL
LIN {X 0,Y 356.264,Z 695.878,A -85,B 0,C 180,E1 15553.562,E2 15553.562} C_VEL
LIN {X 0,Y 359.815,Z 697.671,A -85,B 0,C 180,E1 15559.33,E2 15559.33} C_VEL
LIN {X 0,Y 361.796,Z 698.82,A -85,B 0,C 180,E1 15564.898,E2 15564.898} C_VEL
LIN {X 0,Y 362.261,Z 699.62,A -85,B 0,C 180,E1 15570,E2 15570} C_VEL
LIN {X 0,Y 361.661,Z 698.231,A -85,B 0,C 180,E1 15575.857,E2 15575.857} C_VEL
LIN {X 0,Y 358.99,Z 697.41,A -85,B 0,C 180,E1 15582.174,E2 15582.174} C_VEL
LIN {X 0,Y 355.09,Z 694.754,A -85,B 0,C 180,E1 15588.088,E2 15588.088} C_VEL
LIN {X 0,Y 351.069,Z 689.434,A -85,B 0,C 180,E1 15593.142,E2 15593.142} C_VEL
LIN {X 0,Y 345.326,Z 684.752,A -85,B 0,C 180,E1 15598.577,E2 15598.577} C_VEL
LIN {X 0,Y 342.08,Z 680.778,A -85,B 0,C 180,E1 15601.431,E2 15601.431} C_VEL
LIN {X 0,Y 336.381,Z 674.899,A -85,B 0,C 180,E1 15605.882,E2 15605.882} C_VEL
LIN {X 0,Y 328.87,Z 666.913,A -85,B 0,C 180,E1 15611.19,E2 15611.19} C_VEL
LIN {X 0,Y 321.213,Z 658.418,A -85,B 0,C 180,E1 15616.176,E2 15616.176} C_VEL
LIN {X 0,Y 313.998,Z 650.434,A -85,B 0,C 180,E1 15620.523,E2 15620.523} C_VEL
LIN {X 0,Y 307.239,Z 643.028,A -85,B 0,C 180,E1 15624.263,E2 15624.263} C_VEL
LIN {X 0,Y 300.283,Z 634.275,A -85,B 0,C 180,E1 15627.816,E2 15627.816} C_VEL
LIN {X 0,Y 294.713,Z 627.674,A -85,B 0,C 180,E1 15630.327,E2 15630.327} C_VEL
LIN {X 0,Y 289.366,Z 620.436,A -85,B 0,C 180,E1 15632.716,E2 15632.716} C_VEL
LIN {X 0,Y 284.54,Z 614.035,A -85,B 0,C 180,E1 15635.059,E2 15635.059} C_VEL
LIN {X 0,Y 284.3,Z 611.91,A -85,B 0,C 180,E1 15635.328,E2 15635.328} C_VEL
LIN {X 0,Y 284.665,Z 611.91,A -85,B 0,C 180,E1 15643.21,E2 15643.21} C_VEL
LIN {X 0,Y 285.21,Z 611.91,A -85,B 0,C 180,E1 15651.765,E2 15651.765} C_VEL
LIN {X 0,Y 286.076,Z 611.91,A -85,B 0,C 180,E1 15659.995,E2 15659.995} C_VEL
LIN {X 0,Y 285.501,Z 611.91,A -85,B 0,C 180,E1 15666.083,E2 15666.083} C_VEL
LIN {X 0,Y 285.04,Z 611.91,A -85,B 0,C 180,E1 15672.261,E2 15672.261} C_VEL
LIN {X 0,Y 284.597,Z 611.91,A -85,B 0,C 180,E1 15678.608,E2 15678.608} C_VEL
LIN {X 0,Y 284.303,Z 611.91,A -85,B 0,C 180,E1 15684.264,E2 15684.264} C_VEL
LIN {X 0,Y 286.262,Z 617.203,A -85,B 0,C 180,E1 15685.444,E2 15685.444} C_VEL
LIN {X 0,Y 289.477,Z 620.464,A -85,B 0,C 180,E1 15686.913,E2 15686.913} C_VEL
LIN {X 0,Y 302.879,Z 639.95,A -85,B 0,C 180,E1 15692.416,E2 15692.416} C_VEL
LIN {X 0,Y 316.856,Z 664.058,A -85,B 0,C 180,E1 15697.527,E2 15697.527} C_VEL
LIN {X 0,Y 328.044,Z 689.985,A -85,B 0,C 180,E1 15702.001,E2 15702.001} C_VEL
LIN {X 0,Y 333.592,Z 709.931,A -85,B 0,C 180,E1 15704.955,E2 15704.955} C_VEL
LIN {X 0,Y 324.25,Z 745.731,A -85,B 0,C 180,E1 15708.065,E2 15708.065} C_VEL
LIN {X 0,Y 314.356,Z 776.301,A -85,B 0,C 180,E1 15712.003,E2 15712.003} C_VEL
LIN {X 0,Y 304.83,Z 802.956,A -85,B 0,C 180,E1 15716.883,E2 15716.883} C_VEL
LIN {X 0,Y 296.296,Z 826.121,A -85,B 0,C 180,E1 15722.981,E2 15722.981} C_VEL
LIN {X 0,Y 290.28,Z 844.102,A -85,B 0,C 180,E1 15729.838,E2 15729.838} C_VEL
LIN {X 0,Y 287.336,Z 855.781,A -85,B 0,C 180,E1 15736.677,E2 15736.677} C_VEL
LIN {X 0,Y 286.388,Z 862.876,A -85,B 0,C 180,E1 15743.931,E2 15743.931} C_VEL
LIN {X 0,Y 286.392,Z 864.706,A -85,B 0,C 180,E1 15750,E2 15750} C_VEL
LIN {X 0,Y 286.387,Z 862.876,A -85,B 0,C 180,E1 15756.07,E2 15756.07} C_VEL
LIN {X 0,Y 287.377,Z 855.722,A -85,B 0,C 180,E1 15763.366,E2 15763.366} C_VEL
LIN {X 0,Y 290.586,Z 843.113,A -85,B 0,C 180,E1 15770.64,E2 15770.64} C_VEL
LIN {X 0,Y 297.005,Z 823.908,A -85,B 0,C 180,E1 15777.721,E2 15777.721} C_VEL
LIN {X 0,Y 305.411,Z 801.265,A -85,B 0,C 180,E1 15783.471,E2 15783.471} C_VEL
LIN {X 0,Y 315.689,Z 772.588,A -85,B 0,C 180,E1 15788.571,E2 15788.571} C_VEL
LIN {X 0,Y 325.628,Z 740.672,A -85,B 0,C 180,E1 15792.46,E2 15792.46} C_VEL
LIN {X 0,Y 333.74,Z 709.461,A -85,B 0,C 180,E1 15795.074,E2 15795.074} C_VEL
LIN {X 0,Y 324.617,Z 680.797,A -85,B 0,C 180,E1 15799.486,E2 15799.486} C_VEL
LIN {X 0,Y 314.817,Z 660.163,A -85,B 0,C 180,E1 15803.203,E2 15803.203} C_VEL
LIN {X 0,Y 310.591,Z 656.702,A -85,B 0,C 180,E1 15804.474,E2 15804.474} C_VEL
LIN {X 0,Y 303.757,Z 653.229,A -85,B 0,C 180,E1 15806.545,E2 15806.545} C_VEL
LIN {X 0,Y 303.224,Z 652.4,A -85,B 0,C 180,E1 15806.756,E2 15806.756} C_VEL
LIN {X 0,Y 290.371,Z 632.371,A -85,B 0,C 180,E1 15812.126,E2 15812.126} C_VEL
LIN {X 0,Y 284.75,Z 625.073,A -85,B 0,C 180,E1 15814.741,E2 15814.741} C_VEL
LIN {X 0,Y 280.815,Z 618.99,A -85,B 0,C 180,E1 15816.864,E2 15816.864} C_VEL
LIN {X 0,Y 276.82,Z 614.357,A -85,B 0,C 180,E1 15819.187,E2 15819.187} C_VEL
LIN {X 0,Y 276.447,Z 611.91,A -85,B 0,C 180,E1 15819.8,E2 15819.8} C_VEL
LIN {X 0,Y 277.068,Z 611.91,A -85,B 0,C 180,E1 15827.381,E2 15827.381} C_VEL
LIN {X 0,Y 277.893,Z 611.91,A -85,B 0,C 180,E1 15836.883,E2 15836.883} C_VEL
LIN {X 0,Y 277.93,Z 611.91,A -85,B 0,C 180,E1 15843.128,E2 15843.128} C_VEL
LIN {X 0,Y 277.055,Z 611.91,A -85,B 0,C 180,E1 15852.632,E2 15852.632} C_VEL
LIN {X 0,Y 276.472,Z 612.633,A -85,B 0,C 180,E1 15860.916,E2 15860.916} C_VEL
LIN {X 0,Y 279.083,Z 617.841,A -85,B 0,C 180,E1 15862.637,E2 15862.637} C_VEL
LIN {X 0,Y 281.827,Z 620.399,A -85,B 0,C 180,E1 15864.11,E2 15864.11} C_VEL
LIN {X 0,Y 285.942,Z 626.096,A -85,B 0,C 180,E1 15866.232,E2 15866.232} C_VEL
LIN {X 0,Y 296.861,Z 640.534,A -85,B 0,C 180,E1 15871.309,E2 15871.309} C_VEL
LIN {X 0,Y 307.636,Z 654.01,A -85,B 0,C 180,E1 15876.926,E2 15876.926} C_VEL
LIN {X 0,Y 313.262,Z 659.929,A -85,B 0,C 180,E1 15880.077,E2 15880.077} C_VEL
LIN {X 0,Y 320.34,Z 667.69,A -85,B 0,C 180,E1 15884.35,E2 15884.35} C_VEL
LIN {X 0,Y 327.536,Z 675.479,A -85,B 0,C 180,E1 15889.014,E2 15889.014} C_VEL
LIN {X 0,Y 334.851,Z 683.272,A -85,B 0,C 180,E1 15894.226,E2 15894.226} C_VEL
LIN {X 0,Y 340.873,Z 688.812,A -85,B 0,C 180,E1 15898.849,E2 15898.849} C_VEL
LIN {X 0,Y 346.757,Z 695.57,A -85,B 0,C 180,E1 15904.25,E2 15904.25} C_VEL
LIN {X 0,Y 350.836,Z 698.748,A -85,B 0,C 180,E1 15908.292,E2 15908.292} C_VEL
LIN {X 0,Y 354.807,Z 703.665,A -85,B 0,C 180,E1 15913.605,E2 15913.605} C_VEL
LIN {X 0,Y 358.318,Z 705.423,A -85,B 0,C 180,E1 15919.285,E2 15919.285} C_VEL
LIN {X 0,Y 360.347,Z 706.594,A -85,B 0,C 180,E1 15924.877,E2 15924.877} C_VEL
LIN {X 0,Y 360.798,Z 707.373,A -85,B 0,C 180,E1 15930,E2 15930} C_VEL
LIN {X 0,Y 360.195,Z 706.091,A -85,B 0,C 180,E1 15935.881,E2 15935.881} C_VEL
LIN {X 0,Y 357.664,Z 705.219,A -85,B 0,C 180,E1 15941.908,E2 15941.908} C_VEL
LIN {X 0,Y 353.492,Z 702.475,A -85,B 0,C 180,E1 15948.172,E2 15948.172} C_VEL
LIN {X 0,Y 349.116,Z 696.974,A -85,B 0,C 180,E1 15953.591,E2 15953.591} C_VEL
LIN {X 0,Y 343.337,Z 692.113,A -85,B 0,C 180,E1 15958.939,E2 15958.939} C_VEL
LIN {X 0,Y 340.093,Z 688.284,A -85,B 0,C 180,E1 15961.777,E2 15961.777} C_VEL
LIN {X 0,Y 334.205,Z 681.965,A -85,B 0,C 180,E1 15966.357,E2 15966.357} C_VEL
LIN {X 0,Y 326.813,Z 674.365,A -85,B 0,C 180,E1 15971.495,E2 15971.495} C_VEL
LIN {X 0,Y 318.982,Z 665.696,A -85,B 0,C 180,E1 15976.556,E2 15976.556} C_VEL
LIN {X 0,Y 311.561,Z 657.598,A -85,B 0,C 180,E1 15980.957,E2 15980.957} C_VEL
LIN {X 0,Y 304.548,Z 649.839,A -85,B 0,C 180,E1 15984.809,E2 15984.809} C_VEL
LIN {X 0,Y 293.835,Z 637.446,A -85,B 0,C 180,E1 15990.05,E2 15990.05} C_VEL
LIN {X 0,Y 284.984,Z 625.367,A -85,B 0,C 180,E1 15994.21,E2 15994.21} C_VEL
LIN {X 0,Y 280.631,Z 618.897,A -85,B 0,C 180,E1 15996.542,E2 15996.542} C_VEL
LIN {X 0,Y 276.758,Z 614.024,A -85,B 0,C 180,E1 15998.829,E2 15998.829} C_VEL
LIN {X 0,Y 276.487,Z 611.91,A -85,B 0,C 180,E1 15999.262,E2 15999.262} C_VEL
LIN {X 0,Y 276.982,Z 611.91,A -85,B 0,C 180,E1 16007.365,E2 16007.365} C_VEL
LIN {X 0,Y 277.546,Z 611.91,A -85,B 0,C 180,E1 16013.731,E2 16013.731} C_VEL
LIN {X 0,Y 278.169,Z 611.91,A -85,B 0,C 180,E1 16019.994,E2 16019.994} C_VEL
LIN {X 0,Y 277.558,Z 611.91,A -85,B 0,C 180,E1 16026.257,E2 16026.257} C_VEL
LIN {X 0,Y 277.07,Z 611.91,A -85,B 0,C 180,E1 16032.619,E2 16032.619} C_VEL
LIN {X 0,Y 276.504,Z 612.685,A -85,B 0,C 180,E1 16040.522,E2 16040.522} C_VEL
LIN {X 0,Y 278.851,Z 617.593,A -85,B 0,C 180,E1 16042.089,E2 16042.089} C_VEL
LIN {X 0,Y 282.041,Z 620.71,A -85,B 0,C 180,E1 16043.812,E2 16043.812} C_VEL
LIN {X 0,Y 292.302,Z 635.408,A -85,B 0,C 180,E1 16048.746,E2 16048.746} C_VEL
LIN {X 0,Y 305.591,Z 656.407,A -85,B 0,C 180,E1 16054.188,E2 16054.188} C_VEL
LIN {X 0,Y 318.431,Z 683.094,A -85,B 0,C 180,E1 16059.437,E2 16059.437} C_VEL
LIN {X 0,Y 326.947,Z 709.608,A -85,B 0,C 180,E1 16063.771,E2 16063.771} C_VEL
LIN {X 0,Y 326.898,Z 714.363,A -85,B 0,C 180,E1 16064.32,E2 16064.32} C_VEL
LIN {X 0,Y 317.583,Z 748.05,A -85,B 0,C 180,E1 16067.375,E2 16067.375} C_VEL
LIN {X 0,Y 306.574,Z 780.172,A -85,B 0,C 180,E1 16071.733,E2 16071.733} C_VEL
LIN {X 0,Y 296.842,Z 805.808,A -85,B 0,C 180,E1 16076.747,E2 16076.747} C_VEL
LIN {X 0,Y 287.796,Z 829.456,A -85,B 0,C 180,E1 16083.408,E2 16083.408} C_VEL
LIN {X 0,Y 282.12,Z 845.717,A -85,B 0,C 180,E1 16090.225,E2 16090.225} C_VEL
LIN {X 0,Y 279.245,Z 857.083,A -85,B 0,C 180,E1 16097.474,E2 16097.474} C_VEL
LIN {X 0,Y 278.49,Z 862.641,A -85,B 0,C 180,E1 16103.758,E2 16103.758} C_VEL
LIN {X 0,Y 278.491,Z 864.472,A -85,B 0,C 180,E1 16110,E2 16110} C_VEL
LIN {X 0,Y 278.49,Z 862.641,A -85,B 0,C 180,E1 16116.242,E2 16116.242} C_VEL
LIN {X 0,Y 279.307,Z 856.875,A -85,B 0,C 180,E1 16122.684,E2 16122.684} C_VEL
LIN {X 0,Y 282.691,Z 843.862,A -85,B 0,C 180,E1 16130.728,E2 16130.728} C_VEL
LIN {X 0,Y 288.918,Z 826.242,A -85,B 0,C 180,E1 16137.637,E2 16137.637} C_VEL
LIN {X 0,Y 298.077,Z 802.716,A -85,B 0,C 180,E1 16143.968,E2 16143.968} C_VEL
LIN {X 0,Y 309.029,Z 773.425,A -85,B 0,C 180,E1 16149.333,E2 16149.333} C_VEL
LIN {X 0,Y 319.181,Z 742.423,A -85,B 0,C 180,E1 16153.224,E2 16153.224} C_VEL
LIN {X 0,Y 327.218,Z 710.664,A -85,B 0,C 180,E1 16156.057,E2 16156.057} C_VEL
LIN {X 0,Y 318.427,Z 683.064,A -85,B 0,C 180,E1 16160.566,E2 16160.566} C_VEL
LIN {X 0,Y 305.397,Z 655.989,A -85,B 0,C 180,E1 16165.894,E2 16165.894} C_VEL
LIN {X 0,Y 303.224,Z 652.4,A -85,B 0,C 180,E1 16166.756,E2 16166.756} C_VEL
LIN {X 0,Y 297.957,Z 646.485,A -85,B 0,C 180,E1 16168.743,E2 16168.743} C_VEL
LIN {X 0,Y 288.316,Z 639.839,A -85,B 0,C 180,E1 16172.439,E2 16172.439} C_VEL
LIN {X 0,Y 278.155,Z 625.96,A -85,B 0,C 180,E1 16177.704,E2 16177.704} C_VEL
LIN {X 0,Y 274.252,Z 620.03,A -85,B 0,C 180,E1 16180.201,E2 16180.201} C_VEL
LIN {X 0,Y 269.349,Z 614.636,A -85,B 0,C 180,E1 16183.788,E2 16183.788} C_VEL
LIN {X 0,Y 268.937,Z 611.91,A -85,B 0,C 180,E1 16184.496,E2 16184.496} C_VEL
LIN {X 0,Y 269.616,Z 611.91,A -85,B 0,C 180,E1 16193.558,E2 16193.558} C_VEL
LIN {X 0,Y 270.25,Z 611.91,A -85,B 0,C 180,E1 16200.006,E2 16200.006} C_VEL
LIN {X 0,Y 269.633,Z 611.91,A -85,B 0,C 180,E1 16206.454,E2 16206.454} C_VEL
LIN {X 0,Y 268.948,Z 611.91,A -85,B 0,C 180,E1 16215.934,E2 16215.934} C_VEL
LIN {X 0,Y 270.621,Z 617.081,A -85,B 0,C 180,E1 16217.731,E2 16217.731} C_VEL
LIN {X 0,Y 274.399,Z 620.49,A -85,B 0,C 180,E1 16220.333,E2 16220.333} C_VEL
LIN {X 0,Y 278.665,Z 626.307,A -85,B 0,C 180,E1 16222.988,E2 16222.988} C_VEL
LIN {X 0,Y 294.531,Z 647.959,A -85,B 0,C 180,E1 16231.047,E2 16231.047} C_VEL
LIN {X 0,Y 305.503,Z 661.703,A -85,B 0,C 180,E1 16236.823,E2 16236.823} C_VEL
LIN {X 0,Y 311.364,Z 667.988,A -85,B 0,C 180,E1 16240.118,E2 16240.118} C_VEL
LIN {X 0,Y 317.897,Z 675.051,A -85,B 0,C 180,E1 16244.043,E2 16244.043} C_VEL
LIN {X 0,Y 325.413,Z 683.169,A -85,B 0,C 180,E1 16248.892,E2 16248.892} C_VEL
LIN {X 0,Y 332.612,Z 690.698,A -85,B 0,C 180,E1 16253.951,E2 16253.951} C_VEL
LIN {X 0,Y 339.305,Z 696.592,A -85,B 0,C 180,E1 16259.019,E2 16259.019} C_VEL
LIN {X 0,Y 344.586,Z 703.034,A -85,B 0,C 180,E1 16263.935,E2 16263.935} C_VEL
LIN {X 0,Y 348.798,Z 706.326,A -85,B 0,C 180,E1 16268.122,E2 16268.122} C_VEL
LIN {X 0,Y 352.859,Z 711.293,A -85,B 0,C 180,E1 16273.512,E2 16273.512} C_VEL
LIN {X 0,Y 356.344,Z 713.069,A -85,B 0,C 180,E1 16278.976,E2 16278.976} C_VEL
LIN {X 0,Y 358.484,Z 714.131,A -85,B 0,C 180,E1 16284.547,E2 16284.547} C_VEL
LIN {X 0,Y 358.996,Z 715.063,A -85,B 0,C 180,E1 16290,E2 16290} C_VEL
LIN {X 0,Y 358.39,Z 713.685,A -85,B 0,C 180,E1 16296.063,E2 16296.063} C_VEL
LIN {X 0,Y 355.632,Z 712.807,A -85,B 0,C 180,E1 16302.29,E2 16302.29} C_VEL
LIN {X 0,Y 351.537,Z 710.067,A -85,B 0,C 180,E1 16308.309,E2 16308.309} C_VEL
LIN {X 0,Y 347.174,Z 704.603,A -85,B 0,C 180,E1 16313.671,E2 16313.671} C_VEL
LIN {X 0,Y 341.241,Z 699.627,A -85,B 0,C 180,E1 16319.132,E2 16319.132} C_VEL
LIN {X 0,Y 337.712,Z 695.627,A -85,B 0,C 180,E1 16322.168,E2 16322.168} C_VEL
LIN {X 0,Y 331.731,Z 688.983,A -85,B 0,C 180,E1 16326.825,E2 16326.825} C_VEL
LIN {X 0,Y 324.508,Z 681.749,A -85,B 0,C 180,E1 16331.784,E2 16331.784} C_VEL
LIN {X 0,Y 316.363,Z 672.756,A -85,B 0,C 180,E1 16336.98,E2 16336.98} C_VEL
LIN {X 0,Y 308.922,Z 664.71,A -85,B 0,C 180,E1 16341.365,E2 16341.365} C_VEL
LIN {X 0,Y 301.733,Z 656.822,A -85,B 0,C 180,E1 16345.27,E2 16345.27} C_VEL
LIN {X 0,Y 290.588,Z 643.736,A -85,B 0,C 180,E1 16350.755,E2 16350.755} C_VEL
LIN {X 0,Y 278.168,Z 625.971,A -85,B 0,C 180,E1 16357.281,E2 16357.281} C_VEL
LIN {X 0,Y 274.354,Z 620.197,A -85,B 0,C 180,E1 16359.715,E2 16359.715} C_VEL
LIN {X 0,Y 269.305,Z 614.645,A -85,B 0,C 180,E1 16363.403,E2 16363.403} C_VEL
LIN {X 0,Y 268.912,Z 611.91,A -85,B 0,C 180,E1 16364.064,E2 16364.064} C_VEL
LIN {X 0,Y 269.619,Z 611.91,A -85,B 0,C 180,E1 16373.546,E2 16373.546} C_VEL
LIN {X 0,Y 270.286,Z 611.91,A -85,B 0,C 180,E1 16379.994,E2 16379.994} C_VEL
LIN {X 0,Y 269.631,Z 611.91,A -85,B 0,C 180,E1 16386.442,E2 16386.442} C_VEL
LIN {X 0,Y 268.968,Z 612.279,A -85,B 0,C 180,E1 16395.711,E2 16395.711} C_VEL
LIN {X 0,Y 270.648,Z 617.071,A -85,B 0,C 180,E1 16397.332,E2 16397.332} C_VEL
LIN {X 0,Y 274.386,Z 620.411,A -85,B 0,C 180,E1 16399.904,E2 16399.904} C_VEL
LIN {X 0,Y 278.302,Z 626.082,A -85,B 0,C 180,E1 16402.378,E2 16402.378} C_VEL
LIN {X 0,Y 288.719,Z 640.753,A -85,B 0,C 180,E1 16407.782,E2 16407.782} C_VEL
LIN {X 0,Y 302.025,Z 663.035,A -85,B 0,C 180,E1 16413.673,E2 16413.673} C_VEL
LIN {X 0,Y 313.526,Z 688.445,A -85,B 0,C 180,E1 16418.879,E2 16418.879} C_VEL
LIN {X 0,Y 320.977,Z 713.419,A -85,B 0,C 180,E1 16423.143,E2 16423.143} C_VEL
LIN {X 0,Y 311.61,Z 748.186,A -85,B 0,C 180,E1 16426.422,E2 16426.422} C_VEL
LIN {X 0,Y 300.455,Z 779.56,A -85,B 0,C 180,E1 16430.725,E2 16430.725} C_VEL
LIN {X 0,Y 290.331,Z 805.095,A -85,B 0,C 180,E1 16435.758,E2 16435.758} C_VEL
LIN {X 0,Y 281.034,Z 828.076,A -85,B 0,C 180,E1 16442.288,E2 16442.288} C_VEL
LIN {X 0,Y 274.525,Z 845.427,A -85,B 0,C 180,E1 16449.626,E2 16449.626} C_VEL
LIN {X 0,Y 271.467,Z 856.847,A -85,B 0,C 180,E1 16457.109,E2 16457.109} C_VEL
LIN {X 0,Y 270.593,Z 862.406,A -85,B 0,C 180,E1 16463.575,E2 16463.575} C_VEL
LIN {X 0,Y 270.604,Z 864.239,A -85,B 0,C 180,E1 16470,E2 16470} C_VEL
LIN {X 0,Y 270.592,Z 862.406,A -85,B 0,C 180,E1 16476.425,E2 16476.425} C_VEL
LIN {X 0,Y 271.633,Z 855.816,A -85,B 0,C 180,E1 16483.703,E2 16483.703} C_VEL
LIN {X 0,Y 275.172,Z 843.568,A -85,B 0,C 180,E1 16491.353,E2 16491.353} C_VEL
LIN {X 0,Y 281.788,Z 825.807,A -85,B 0,C 180,E1 16498.471,E2 16498.471} C_VEL
LIN {X 0,Y 291.385,Z 802.476,A -85,B 0,C 180,E1 16504.86,E2 16504.86} C_VEL
LIN {X 0,Y 302.863,Z 773.177,A -85,B 0,C 180,E1 16510.298,E2 16510.298} C_VEL
LIN {X 0,Y 313.39,Z 742.186,A -85,B 0,C 180,E1 16514.227,E2 16514.227} C_VEL
LIN {X 0,Y 321.003,Z 713.44,A -85,B 0,C 180,E1 16516.85,E2 16516.85} C_VEL
LIN {X 0,Y 312.851,Z 686.872,A -85,B 0,C 180,E1 16521.425,E2 16521.425} C_VEL
LIN {X 0,Y 301.022,Z 661.267,A -85,B 0,C 180,E1 16526.74,E2 16526.74} C_VEL
LIN {X 0,Y 288.316,Z 639.839,A -85,B 0,C 180,E1 16532.439,E2 16532.439} C_VEL
LIN {X 0,Y 275.074,Z 632.219,A -85,B 0,C 180,E1 16538.863,E2 16538.863} C_VEL
LIN {X 0,Y 271.07,Z 626.34,A -85,B 0,C 180,E1 16541.618,E2 16541.618} C_VEL
LIN {X 0,Y 267.399,Z 621.203,A -85,B 0,C 180,E1 16544.615,E2 16544.615} C_VEL
LIN {X 0,Y 266.385,Z 619.362,A -85,B 0,C 180,E1 16545.608,E2 16545.608} C_VEL
LIN {X 0,Y 261.947,Z 614.703,A -85,B 0,C 180,E1 16550.71,E2 16550.71} C_VEL
LIN {X 0,Y 261.515,Z 611.91,A -85,B 0,C 180,E1 16552.103,E2 16552.103} C_VEL
LIN {X 0,Y 262.343,Z 611.91,A -85,B 0,C 180,E1 16560.006,E2 16560.006} C_VEL
LIN {X 0,Y 261.475,Z 612.336,A -85,B 0,C 180,E1 16568.644,E2 16568.644} C_VEL
LIN {X 0,Y 263.586,Z 617.595,A -85,B 0,C 180,E1 16572.024,E2 16572.024} C_VEL
LIN {X 0,Y 267.149,Z 620.473,A -85,B 0,C 180,E1 16575.535,E2 16575.535} C_VEL
LIN {X 0,Y 270.285,Z 625.782,A -85,B 0,C 180,E1 16578.249,E2 16578.249} C_VEL
LIN {X 0,Y 272.698,Z 628.5,A -85,B 0,C 180,E1 16579.98,E2 16579.98} C_VEL
LIN {X 0,Y 278.337,Z 636.993,A -85,B 0,C 180,E1 16583.657,E2 16583.657} C_VEL
LIN {X 0,Y 295.202,Z 660.053,A -85,B 0,C 180,E1 16592.503,E2 16592.503} C_VEL
LIN {X 0,Y 305.487,Z 671.169,A -85,B 0,C 180,E1 16597.937,E2 16597.937} C_VEL
LIN {X 0,Y 315.72,Z 682.91,A -85,B 0,C 180,E1 16604.057,E2 16604.057} C_VEL
LIN {X 0,Y 322.822,Z 690.489,A -85,B 0,C 180,E1 16608.631,E2 16608.631} C_VEL
LIN {X 0,Y 330.009,Z 697.959,A -85,B 0,C 180,E1 16613.65,E2 16613.65} C_VEL
LIN {X 0,Y 338.219,Z 706.115,A -85,B 0,C 180,E1 16620.071,E2 16620.071} C_VEL
LIN {X 0,Y 342.188,Z 710.46,A -85,B 0,C 180,E1 16623.739,E2 16623.739} C_VEL
LIN {X 0,Y 346.468,Z 713.892,A -85,B 0,C 180,E1 16627.997,E2 16627.997} C_VEL
LIN {X 0,Y 349.787,Z 718.194,A -85,B 0,C 180,E1 16632.362,E2 16632.362} C_VEL
LIN {X 0,Y 353.973,Z 720.572,A -85,B 0,C 180,E1 16638.546,E2 16638.546} C_VEL
LIN {X 0,Y 356.321,Z 721.632,A -85,B 0,C 180,E1 16644.325,E2 16644.325} C_VEL
LIN {X 0,Y 356.87,Z 722.643,A -85,B 0,C 180,E1 16650,E2 16650} C_VEL
LIN {X 0,Y 356.274,Z 721.367,A -85,B 0,C 180,E1 16655.992,E2 16655.992} C_VEL
LIN {X 0,Y 353.919,Z 720.581,A -85,B 0,C 180,E1 16661.455,E2 16661.455} C_VEL
LIN {X 0,Y 349.793,Z 718.15,A -85,B 0,C 180,E1 16667.637,E2 16667.637} C_VEL
LIN {X 0,Y 345.521,Z 712.407,A -85,B 0,C 180,E1 16673.227,E2 16673.227} C_VEL
LIN {X 0,Y 339.043,Z 707.398,A -85,B 0,C 180,E1 16679.113,E2 16679.113} C_VEL
LIN {X 0,Y 335.542,Z 703.241,A -85,B 0,C 180,E1 16682.185,E2 16682.185} C_VEL
LIN {X 0,Y 329.239,Z 696.45,A -85,B 0,C 180,E1 16687.029,E2 16687.029} C_VEL
LIN {X 0,Y 321.71,Z 688.79,A -85,B 0,C 180,E1 16692.18,E2 16692.18} C_VEL
LIN {X 0,Y 313.679,Z 680.114,A -85,B 0,C 180,E1 16697.263,E2 16697.263} C_VEL
LIN {X 0,Y 302.619,Z 668.941,A -85,B 0,C 180,E1 16703.52,E2 16703.52} C_VEL
LIN {X 0,Y 291.017,Z 654.529,A -85,B 0,C 180,E1 16709.622,E2 16709.622} C_VEL
LIN {X 0,Y 275.615,Z 632.896,A -85,B 0,C 180,E1 16718.018,E2 16718.018} C_VEL
LIN {X 0,Y 271.324,Z 626.479,A -85,B 0,C 180,E1 16721.033,E2 16721.033} C_VEL
LIN {X 0,Y 267.441,Z 621.549,A -85,B 0,C 180,E1 16724.133,E2 16724.133} C_VEL
LIN {X 0,Y 266.404,Z 619.379,A -85,B 0,C 180,E1 16725.175,E2 16725.175} C_VEL
LIN {X 0,Y 261.98,Z 614.876,A -85,B 0,C 180,E1 16730.222,E2 16730.222} C_VEL
LIN {X 0,Y 261.459,Z 611.91,A -85,B 0,C 180,E1 16731.845,E2 16731.845} C_VEL
LIN {X 0,Y 262.378,Z 611.91,A -85,B 0,C 180,E1 16739.994,E2 16739.994} C_VEL
LIN {X 0,Y 261.514,Z 612.507,A -85,B 0,C 180,E1 16748.316,E2 16748.316} C_VEL
LIN {X 0,Y 263.927,Z 617.899,A -85,B 0,C 180,E1 16751.996,E2 16751.996} C_VEL
LIN {X 0,Y 267.225,Z 620.538,A -85,B 0,C 180,E1 16755.185,E2 16755.185} C_VEL
LIN {X 0,Y 270.633,Z 626.049,A -85,B 0,C 180,E1 16758.08,E2 16758.08} C_VEL
LIN {X 0,Y 272.733,Z 628.577,A -85,B 0,C 180,E1 16759.565,E2 16759.565} C_VEL
LIN {X 0,Y 278.452,Z 636.872,A -85,B 0,C 180,E1 16763.21,E2 16763.21} C_VEL
LIN {X 0,Y 286.757,Z 649.105,A -85,B 0,C 180,E1 16767.615,E2 16767.615} C_VEL
LIN {X 0,Y 298.377,Z 669.899,A -85,B 0,C 180,E1 16773.267,E2 16773.267} C_VEL
LIN {X 0,Y 309.026,Z 695.134,A -85,B 0,C 180,E1 16778.561,E2 16778.561} C_VEL
LIN {X 0,Y 314.983,Z 717.644,A -85,B 0,C 180,E1 16782.531,E2 16782.531} C_VEL
LIN {X 0,Y 305.38,Z 749.297,A -85,B 0,C 180,E1 16785.548,E2 16785.548} C_VEL
LIN {X 0,Y 293.424,Z 781.448,A -85,B 0,C 180,E1 16790.076,E2 16790.076} C_VEL
LIN {X 0,Y 282.128,Z 808.344,A -85,B 0,C 180,E1 16795.703,E2 16795.703} C_VEL
LIN {X 0,Y 272.851,Z 830.227,A -85,B 0,C 180,E1 16802.365,E2 16802.365} C_VEL
LIN {X 0,Y 266.331,Z 847.091,A -85,B 0,C 180,E1 16810.057,E2 16810.057} C_VEL
LIN {X 0,Y 263.422,Z 857.596,A -85,B 0,C 180,E1 16817.675,E2 16817.675} C_VEL
LIN {X 0,Y 262.696,Z 862.171,A -85,B 0,C 180,E1 16823.381,E2 16823.381} C_VEL
LIN {X 0,Y 262.703,Z 864.005,A -85,B 0,C 180,E1 16830,E2 16830} C_VEL
LIN {X 0,Y 262.696,Z 862.171,A -85,B 0,C 180,E1 16836.619,E2 16836.619} C_VEL
LIN {X 0,Y 263.845,Z 855.578,A -85,B 0,C 180,E1 16844.116,E2 16844.116} C_VEL
LIN {X 0,Y 267.724,Z 843.095,A -85,B 0,C 180,E1 16852.112,E2 16852.112} C_VEL
LIN {X 0,Y 275.21,Z 824.366,A -85,B 0,C 180,E1 16859.678,E2 16859.678} C_VEL
LIN {X 0,Y 284.767,Z 802.237,A -85,B 0,C 180,E1 16865.792,E2 16865.792} C_VEL
LIN {X 0,Y 296.81,Z 772.94,A -85,B 0,C 180,E1 16871.296,E2 16871.296} C_VEL
LIN {X 0,Y 307.732,Z 741.951,A -85,B 0,C 180,E1 16875.262,E2 16875.262} C_VEL
LIN {X 0,Y 314.822,Z 716.156,A -85,B 0,C 180,E1 16877.687,E2 16877.687} C_VEL
LIN {X 0,Y 307.342,Z 690.484,A -85,B 0,C 180,E1 16882.337,E2 16882.337} C_VEL
LIN {X 0,Y 295.9,Z 664.94,A -85,B 0,C 180,E1 16887.944,E2 16887.944} C_VEL
LIN {X 0,Y 284.485,Z 645.504,A -85,B 0,C 180,E1 16893.538,E2 16893.538} C_VEL
LIN {X 0,Y 275.819,Z 632.983,A -85,B 0,C 180,E1 16898.412,E2 16898.412} C_VEL
LIN {X 0,Y 275.074,Z 632.219,A -85,B 0,C 180,E1 16898.863,E2 16898.863} C_VEL
LIN {X 0,Y 267.296,Z 627.95,A -85,B 0,C 180,E1 16904.045,E2 16904.045} C_VEL
LIN {X 0,Y 265.109,Z 627.1,A -85,B 0,C 180,E1 16905.855,E2 16905.855} C_VEL
LIN {X 0,Y 260.66,Z 622.185,A -85,B 0,C 180,E1 16911.189,E2 16911.189} C_VEL
LIN {X 0,Y 260.074,Z 619.652,A -85,B 0,C 180,E1 16912.539,E2 16912.539} C_VEL
LIN {X 0,Y 258.34,Z 618.93,A -85,B 0,C 180,E1 16923.786,E2 16923.786} C_VEL
LIN {X 0,Y 260.263,Z 620.638,A -85,B 0,C 180,E1 16928.37,E2 16928.37} C_VEL
LIN {X 0,Y 263.321,Z 626.063,A -85,B 0,C 180,E1 16932.827,E2 16932.827} C_VEL
LIN {X 0,Y 265.59,Z 628.388,A -85,B 0,C 180,E1 16935.113,E2 16935.113} C_VEL
LIN {X 0,Y 269.623,Z 634.053,A -85,B 0,C 180,E1 16938.631,E2 16938.631} C_VEL
LIN {X 0,Y 278.69,Z 648.211,A -85,B 0,C 180,E1 16944.905,E2 16944.905} C_VEL
LIN {X 0,Y 293.168,Z 668.232,A -85,B 0,C 180,E1 16952.69,E2 16952.69} C_VEL
LIN {X 0,Y 303.971,Z 680.103,A -85,B 0,C 180,E1 16958.512,E2 16958.512} C_VEL
LIN {X 0,Y 313.607,Z 691.118,A -85,B 0,C 180,E1 16964.332,E2 16964.332} C_VEL
LIN {X 0,Y 320.852,Z 698.876,A -85,B 0,C 180,E1 16969.032,E2 16969.032} C_VEL
LIN {X 0,Y 327.671,Z 705.85,A -85,B 0,C 180,E1 16973.811,E2 16973.811} C_VEL
LIN {X 0,Y 334.798,Z 712.404,A -85,B 0,C 180,E1 16979.236,E2 16979.236} C_VEL
LIN {X 0,Y 339.388,Z 717.736,A -85,B 0,C 180,E1 16983.505,E2 16983.505} C_VEL
LIN {X 0,Y 343.748,Z 721.022,A -85,B 0,C 180,E1 16987.668,E2 16987.668} C_VEL
LIN {X 0,Y 347.898,Z 726.145,A -85,B 0,C 180,E1 16993.232,E2 16993.232} C_VEL
LIN {X 0,Y 350.882,Z 727.781,A -85,B 0,C 180,E1 16997.54,E2 16997.54} C_VEL
LIN {X 0,Y 353.481,Z 728.532,A -85,B 0,C 180,E1 17002.617,E2 17002.617} C_VEL
LIN {X 0,Y 354.34,Z 729.834,A -85,B 0,C 180,E1 17007.551,E2 17007.551} C_VEL
LIN {X 0,Y 354.314,Z 730.033,A -85,B 0,C 180,E1 17012.449,E2 17012.449} C_VEL
LIN {X 0,Y 353.456,Z 728.507,A -85,B 0,C 180,E1 17017.383,E2 17017.383} C_VEL
LIN {X 0,Y 350.871,Z 727.845,A -85,B 0,C 180,E1 17022.46,E2 17022.46} C_VEL
LIN {X 0,Y 347.171,Z 725.542,A -85,B 0,C 180,E1 17027.775,E2 17027.775} C_VEL
LIN {X 0,Y 342.851,Z 719.805,A -85,B 0,C 180,E1 17033.419,E2 17033.419} C_VEL
LIN {X 0,Y 336.808,Z 715.33,A -85,B 0,C 180,E1 17038.847,E2 17038.847} C_VEL
LIN {X 0,Y 331.628,Z 709.736,A -85,B 0,C 180,E1 17043.22,E2 17043.22} C_VEL
LIN {X 0,Y 323.734,Z 701.593,A -85,B 0,C 180,E1 17049.053,E2 17049.053} C_VEL
LIN {X 0,Y 316.195,Z 693.559,A -85,B 0,C 180,E1 17054.085,E2 17054.085} C_VEL
LIN {X 0,Y 306.36,Z 683.37,A -85,B 0,C 180,E1 17060.019,E2 17060.019} C_VEL
LIN {X 0,Y 295.5,Z 670.698,A -85,B 0,C 180,E1 17066.123,E2 17066.123} C_VEL
LIN {X 0,Y 283.485,Z 655.948,A -85,B 0,C 180,E1 17072.242,E2 17072.242} C_VEL
LIN {X 0,Y 273.249,Z 639.867,A -85,B 0,C 180,E1 17078.672,E2 17078.672} C_VEL
LIN {X 0,Y 269.064,Z 633.696,A -85,B 0,C 180,E1 17081.754,E2 17081.754} C_VEL
LIN {X 0,Y 265.48,Z 627.98,A -85,B 0,C 180,E1 17085.028,E2 17085.028} C_VEL
LIN {X 0,Y 260.506,Z 621.784,A -85,B 0,C 180,E1 17091.059,E2 17091.059} C_VEL
LIN {X 0,Y 259.924,Z 619.623,A -85,B 0,C 180,E1 17092.379,E2 17092.379} C_VEL
LIN {X 0,Y 258.452,Z 618.997,A -85,B 0,C 180,E1 17103.773,E2 17103.773} C_VEL
LIN {X 0,Y 260.263,Z 620.586,A -85,B 0,C 180,E1 17107.944,E2 17107.944} C_VEL
LIN {X 0,Y 263.348,Z 626.119,A -85,B 0,C 180,E1 17112.444,E2 17112.444} C_VEL
LIN {X 0,Y 265.675,Z 628.385,A -85,B 0,C 180,E1 17114.747,E2 17114.747} C_VEL
LIN {X 0,Y 269.781,Z 634.11,A -85,B 0,C 180,E1 17118.242,E2 17118.242} C_VEL
LIN {X 0,Y 279.61,Z 648.907,A -85,B 0,C 180,E1 17124.699,E2 17124.699} C_VEL
LIN {X 0,Y 290.1,Z 667.394,A -85,B 0,C 180,E1 17130.472,E2 17130.472} C_VEL
LIN {X 0,Y 300.982,Z 691.669,A -85,B 0,C 180,E1 17136.227,E2 17136.227} C_VEL
LIN {X 0,Y 308.325,Z 717.167,A -85,B 0,C 180,E1 17141.14,E2 17141.14} C_VEL
LIN {X 0,Y 308.27,Z 722.421,A -85,B 0,C 180,E1 17141.845,E2 17141.845} C_VEL
LIN {X 0,Y 296.902,Z 756.722,A -85,B 0,C 180,E1 17145.397,E2 17145.397} C_VEL
LIN {X 0,Y 285.199,Z 786.055,A -85,B 0,C 180,E1 17149.933,E2 17149.933} C_VEL
LIN {X 0,Y 273.493,Z 812.564,A -85,B 0,C 180,E1 17155.908,E2 17155.908} C_VEL
LIN {X 0,Y 263.911,Z 833.975,A -85,B 0,C 180,E1 17163.142,E2 17163.142} C_VEL
LIN {X 0,Y 258.253,Z 848.309,A -85,B 0,C 180,E1 17170.299,E2 17170.299} C_VEL
LIN {X 0,Y 255.524,Z 857.674,A -85,B 0,C 180,E1 17177.632,E2 17177.632} C_VEL
LIN {X 0,Y 254.807,Z 861.937,A -85,B 0,C 180,E1 17183.175,E2 17183.175} C_VEL
LIN {X 0,Y 254.818,Z 863.772,A -85,B 0,C 180,E1 17190,E2 17190} C_VEL
LIN {X 0,Y 254.806,Z 861.937,A -85,B 0,C 180,E1 17196.825,E2 17196.825} C_VEL
LIN {X 0,Y 256.08,Z 855.342,A -85,B 0,C 180,E1 17204.553,E2 17204.553} C_VEL
LIN {X 0,Y 260.462,Z 842.427,A -85,B 0,C 180,E1 17213.012,E2 17213.012} C_VEL
LIN {X 0,Y 268.774,Z 822.951,A -85,B 0,C 180,E1 17220.933,E2 17220.933} C_VEL
LIN {X 0,Y 278.862,Z 800.572,A -85,B 0,C 180,E1 17227.082,E2 17227.082} C_VEL
LIN {X 0,Y 291.266,Z 771.639,A -85,B 0,C 180,E1 17232.513,E2 17232.513} C_VEL
LIN {X 0,Y 302.636,Z 740.185,A -85,B 0,C 180,E1 17236.504,E2 17236.504} C_VEL
LIN {X 0,Y 308.958,Z 720.186,A -85,B 0,C 180,E1 17238.336,E2 17238.336} C_VEL
LIN {X 0,Y 302.176,Z 695.202,A -85,B 0,C 180,E1 17243.048,E2 17243.048} C_VEL
LIN {X 0,Y 291.143,Z 669.211,A -85,B 0,C 180,E1 17248.999,E2 17248.999} C_VEL
LIN {X 0,Y 280.648,Z 650.892,A -85,B 0,C 180,E1 17254.653,E2 17254.653} C_VEL
LIN {X 0,Y 273.243,Z 639.684,A -85,B 0,C 180,E1 17259.215,E2 17259.215} C_VEL
LIN {X 0,Y 268.979,Z 633.516,A -85,B 0,C 180,E1 17262.342,E2 17262.342} C_VEL
LIN {X 0,Y 265.501,Z 627.801,A -85,B 0,C 180,E1 17265.454,E2 17265.454} C_VEL
LIN {X 0,Y 265.109,Z 627.1,A -85,B 0,C 180,E1 17265.855,E2 17265.855} C_VEL
LIN {X 0,Y 258.678,Z 627.371,A -85,B 0,C 180,E1 17273.301,E2 17273.301} C_VEL
LIN {X 0,Y 257.493,Z 626.869,A -85,B 0,C 180,E1 17284.221,E2 17284.221} C_VEL
LIN {X 0,Y 259.06,Z 628.373,A -85,B 0,C 180,E1 17287.986,E2 17287.986} C_VEL
LIN {X 0,Y 262.084,Z 633.886,A -85,B 0,C 180,E1 17292.729,E2 17292.729} C_VEL
LIN {X 0,Y 263.959,Z 636.199,A -85,B 0,C 180,E1 17294.751,E2 17294.751} C_VEL
LIN {X 0,Y 268.921,Z 644.021,A -85,B 0,C 180,E1 17299.321,E2 17299.321} C_VEL
LIN {X 0,Y 275.972,Z 655.583,A -85,B 0,C 180,E1 17304.518,E2 17304.518} C_VEL
LIN {X 0,Y 289.858,Z 675.222,A -85,B 0,C 180,E1 17312.377,E2 17312.377} C_VEL
LIN {X 0,Y 300.512,Z 686.891,A -85,B 0,C 180,E1 17318.116,E2 17318.116} C_VEL
LIN {X 0,Y 309.781,Z 697.415,A -85,B 0,C 180,E1 17323.672,E2 17323.672} C_VEL
LIN {X 0,Y 317.728,Z 706.017,A -85,B 0,C 180,E1 17328.827,E2 17328.827} C_VEL
LIN {X 0,Y 325.812,Z 714.459,A -85,B 0,C 180,E1 17334.553,E2 17334.553} C_VEL
LIN {X 0,Y 332.674,Z 721.11,A -85,B 0,C 180,E1 17339.958,E2 17339.958} C_VEL
LIN {X 0,Y 337.085,Z 725.442,A -85,B 0,C 180,E1 17343.944,E2 17343.944} C_VEL
LIN {X 0,Y 340.764,Z 728.209,A -85,B 0,C 180,E1 17347.462,E2 17347.462} C_VEL
LIN {X 0,Y 344.237,Z 732.865,A -85,B 0,C 180,E1 17352.068,E2 17352.068} C_VEL
LIN {X 0,Y 348.008,Z 735.126,A -85,B 0,C 180,E1 17357.436,E2 17357.436} C_VEL
LIN {X 0,Y 350.792,Z 736.112,A -85,B 0,C 180,E1 17363.092,E2 17363.092} C_VEL
LIN {X 0,Y 351.564,Z 737.225,A -85,B 0,C 180,E1 17367.532,E2 17367.532} C_VEL
LIN {X 0,Y 351.529,Z 737.416,A -85,B 0,C 180,E1 17372.468,E2 17372.468} C_VEL
LIN {X 0,Y 350.693,Z 735.897,A -85,B 0,C 180,E1 17377.442,E2 17377.442} C_VEL
LIN {X 0,Y 347.982,Z 735.183,A -85,B 0,C 180,E1 17382.565,E2 17382.565} C_VEL
LIN {X 0,Y 344.225,Z 732.817,A -85,B 0,C 180,E1 17387.932,E2 17387.932} C_VEL
LIN {X 0,Y 339.801,Z 727.05,A -85,B 0,C 180,E1 17393.642,E2 17393.642} C_VEL
LIN {X 0,Y 333.683,Z 722.369,A -85,B 0,C 180,E1 17399.143,E2 17399.143} C_VEL
LIN {X 0,Y 328.034,Z 716.503,A -85,B 0,C 180,E1 17403.814,E2 17403.814} C_VEL
LIN {X 0,Y 320.356,Z 708.498,A -85,B 0,C 180,E1 17409.455,E2 17409.455} C_VEL
LIN {X 0,Y 311.584,Z 699.347,A -85,B 0,C 180,E1 17415.199,E2 17415.199} C_VEL
LIN {X 0,Y 301.66,Z 688.765,A -85,B 0,C 180,E1 17421.138,E2 17421.138} C_VEL
LIN {X 0,Y 289.858,Z 675.295,A -85,B 0,C 180,E1 17427.623,E2 17427.623} C_VEL
LIN {X 0,Y 272.254,Z 648.967,A -85,B 0,C 180,E1 17438.162,E2 17438.162} C_VEL
LIN {X 0,Y 266.875,Z 640.842,A -85,B 0,C 180,E1 17442.453,E2 17442.453} C_VEL
LIN {X 0,Y 262.823,Z 634.437,A -85,B 0,C 180,E1 17446.46,E2 17446.46} C_VEL
LIN {X 0,Y 259.238,Z 629.315,A -85,B 0,C 180,E1 17451.516,E2 17451.516} C_VEL
LIN {X 0,Y 258.479,Z 627.335,A -85,B 0,C 180,E1 17453.266,E2 17453.266} C_VEL
LIN {X 0,Y 257.49,Z 626.847,A -85,B 0,C 180,E1 17463.787,E2 17463.787} C_VEL
LIN {X 0,Y 259.067,Z 628.416,A -85,B 0,C 180,E1 17467.588,E2 17467.588} C_VEL
LIN {X 0,Y 262.515,Z 634.148,A -85,B 0,C 180,E1 17472.696,E2 17472.696} C_VEL
LIN {X 0,Y 264.201,Z 636.543,A -85,B 0,C 180,E1 17474.513,E2 17474.513} C_VEL
LIN {X 0,Y 269.299,Z 644.287,A -85,B 0,C 180,E1 17478.961,E2 17478.961} C_VEL
LIN {X 0,Y 276.573,Z 655.41,A -85,B 0,C 180,E1 17484.019,E2 17484.019} C_VEL
LIN {X 0,Y 287.245,Z 675.367,A -85,B 0,C 180,E1 17490.368,E2 17490.368} C_VEL
LIN {X 0,Y 296.857,Z 699.526,A -85,B 0,C 180,E1 17496.164,E2 17496.164} C_VEL
LIN {X 0,Y 302.715,Z 723.099,A -85,B 0,C 180,E1 17500.801,E2 17500.801} C_VEL
LIN {X 0,Y 290.751,Z 757.867,A -85,B 0,C 180,E1 17504.463,E2 17504.463} C_VEL
LIN {X 0,Y 278.22,Z 787.713,A -85,B 0,C 180,E1 17509.229,E2 17509.229} C_VEL
LIN {X 0,Y 266.843,Z 812.326,A -85,B 0,C 180,E1 17514.936,E2 17514.936} C_VEL
LIN {X 0,Y 257.005,Z 833.114,A -85,B 0,C 180,E1 17522.071,E2 17522.071} C_VEL
LIN {X 0,Y 250.644,Z 848.15,A -85,B 0,C 180,E1 17529.733,E2 17529.733} C_VEL
LIN {X 0,Y 247.522,Z 858.224,A -85,B 0,C 180,E1 17538.11,E2 17538.11} C_VEL
LIN {X 0,Y 246.913,Z 861.702,A -85,B 0,C 180,E1 17542.956,E2 17542.956} C_VEL
LIN {X 0,Y 246.915,Z 863.539,A -85,B 0,C 180,E1 17550,E2 17550} C_VEL
LIN {X 0,Y 246.913,Z 861.702,A -85,B 0,C 180,E1 17557.044,E2 17557.044} C_VEL
LIN {X 0,Y 248.32,Z 855.104,A -85,B 0,C 180,E1 17565.018,E2 17565.018} C_VEL
LIN {X 0,Y 253.116,Z 842.023,A -85,B 0,C 180,E1 17573.814,E2 17573.814} C_VEL
LIN {X 0,Y 261.817,Z 822.815,A -85,B 0,C 180,E1 17581.807,E2 17581.807} C_VEL
LIN {X 0,Y 272.34,Z 800.573,A -85,B 0,C 180,E1 17588.055,E2 17588.055} C_VEL
LIN {X 0,Y 285.353,Z 771.4,A -85,B 0,C 180,E1 17593.612,E2 17593.612} C_VEL
LIN {X 0,Y 297.173,Z 739.948,A -85,B 0,C 180,E1 17597.626,E2 17597.626} C_VEL
LIN {X 0,Y 302.606,Z 721.736,A -85,B 0,C 180,E1 17599.434,E2 17599.434} C_VEL
LIN {X 0,Y 296.205,Z 697.519,A -85,B 0,C 180,E1 17604.268,E2 17604.268} C_VEL
LIN {X 0,Y 286.088,Z 673.071,A -85,B 0,C 180,E1 17610.272,E2 17610.272} C_VEL
LIN {X 0,Y 275.851,Z 654.141,A -85,B 0,C 180,E1 17616.451,E2 17616.451} C_VEL
LIN {X 0,Y 267.252,Z 641.041,A -85,B 0,C 180,E1 17622.704,E2 17622.704} C_VEL
LIN {X 0,Y 262.925,Z 634.368,A -85,B 0,C 180,E1 17626.901,E2 17626.901} C_VEL
LIN {X 0,Y 259.184,Z 628.947,A -85,B 0,C 180,E1 17632.121,E2 17632.121} C_VEL
LIN {X 0,Y 258.678,Z 627.371,A -85,B 0,C 180,E1 17633.301,E2 17633.301} C_VEL
LIN {X 0,Y 256.769,Z 630.562,A -85,B 0,C 180,E1 17637.111,E2 17637.111} C_VEL
LIN {X 0,Y 255.863,Z 634.217,A -85,B 0,C 180,E1 17640.961,E2 17640.961} C_VEL
LIN {X 0,Y 257.732,Z 636.187,A -85,B 0,C 180,E1 17647.707,E2 17647.707} C_VEL
LIN {X 0,Y 260.887,Z 641.75,A -85,B 0,C 180,E1 17652.789,E2 17652.789} C_VEL
LIN {X 0,Y 262.507,Z 644.786,A -85,B 0,C 180,E1 17654.835,E2 17654.835} C_VEL
LIN {X 0,Y 266.719,Z 651.489,A -85,B 0,C 180,E1 17658.949,E2 17658.949} C_VEL
LIN {X 0,Y 273.635,Z 663.941,A -85,B 0,C 180,E1 17664.524,E2 17664.524} C_VEL
LIN {X 0,Y 290.086,Z 686.643,A -85,B 0,C 180,E1 17674.104,E2 17674.104} C_VEL
LIN {X 0,Y 301.895,Z 699.238,A -85,B 0,C 180,E1 17680.695,E2 17680.695} C_VEL
LIN {X 0,Y 312.504,Z 710.56,A -85,B 0,C 180,E1 17687.29,E2 17687.29} C_VEL
LIN {X 0,Y 321.066,Z 719.817,A -85,B 0,C 180,E1 17693.295,E2 17693.295} C_VEL
LIN {X 0,Y 329.205,Z 727.9,A -85,B 0,C 180,E1 17699.609,E2 17699.609} C_VEL
LIN {X 0,Y 334.851,Z 733.241,A -85,B 0,C 180,E1 17704.737,E2 17704.737} C_VEL
LIN {X 0,Y 339.205,Z 738.126,A -85,B 0,C 180,E1 17709.617,E2 17709.617} C_VEL
LIN {X 0,Y 343.745,Z 741.862,A -85,B 0,C 180,E1 17715.708,E2 17715.708} C_VEL
LIN {X 0,Y 346.394,Z 742.964,A -85,B 0,C 180,E1 17719.931,E2 17719.931} C_VEL
LIN {X 0,Y 348.075,Z 744.131,A -85,B 0,C 180,E1 17725.009,E2 17725.009} C_VEL
LIN {X 0,Y 348.542,Z 744.767,A -85,B 0,C 180,E1 17730,E2 17730} C_VEL
LIN {X 0,Y 348.185,Z 744.054,A -85,B 0,C 180,E1 17734.989,E2 17734.989} C_VEL
LIN {X 0,Y 346.355,Z 742.891,A -85,B 0,C 180,E1 17740.07,E2 17740.07} C_VEL
LIN {X 0,Y 342.935,Z 741.469,A -85,B 0,C 180,E1 17745.361,E2 17745.361} C_VEL
LIN {X 0,Y 338.753,Z 737.502,A -85,B 0,C 180,E1 17750.95,E2 17750.95} C_VEL
LIN {X 0,Y 334.885,Z 733.245,A -85,B 0,C 180,E1 17755.275,E2 17755.275} C_VEL
LIN {X 0,Y 329.211,Z 727.871,A -85,B 0,C 180,E1 17760.391,E2 17760.391} C_VEL
LIN {X 0,Y 321.12,Z 719.699,A -85,B 0,C 180,E1 17766.718,E2 17766.718} C_VEL
LIN {X 0,Y 311.771,Z 709.51,A -85,B 0,C 180,E1 17773.239,E2 17773.239} C_VEL
LIN {X 0,Y 300.857,Z 698.503,A -85,B 0,C 180,E1 17779.847,E2 17779.847} C_VEL
LIN {X 0,Y 290.006,Z 686.777,A -85,B 0,C 180,E1 17785.893,E2 17785.893} C_VEL
LIN {X 0,Y 273.367,Z 663.474,A -85,B 0,C 180,E1 17795.669,E2 17795.669} C_VEL
LIN {X 0,Y 266.839,Z 651.647,A -85,B 0,C 180,E1 17800.953,E2 17800.953} C_VEL
LIN {X 0,Y 263.896,Z 647.289,A -85,B 0,C 180,E1 17803.645,E2 17803.645} C_VEL
LIN {X 0,Y 261.054,Z 641.954,A -85,B 0,C 180,E1 17807.007,E2 17807.007} C_VEL
LIN {X 0,Y 257.723,Z 636.444,A -85,B 0,C 180,E1 17812.186,E2 17812.186} C_VEL
LIN {X 0,Y 256.638,Z 634.849,A -85,B 0,C 180,E1 17814.917,E2 17814.917} C_VEL
LIN {X 0,Y 256.526,Z 634.766,A -85,B 0,C 180,E1 17824.225,E2 17824.225} C_VEL
LIN {X 0,Y 257.782,Z 636.36,A -85,B 0,C 180,E1 17827.375,E2 17827.375} C_VEL
LIN {X 0,Y 261.345,Z 642.023,A -85,B 0,C 180,E1 17832.753,E2 17832.753} C_VEL
LIN {X 0,Y 267.156,Z 651.753,A -85,B 0,C 180,E1 17838.582,E2 17838.582} C_VEL
LIN {X 0,Y 274.044,Z 663.105,A -85,B 0,C 180,E1 17843.713,E2 17843.713} C_VEL
LIN {X 0,Y 283.401,Z 681.849,A -85,B 0,C 180,E1 17849.875,E2 17849.875} C_VEL
LIN {X 0,Y 292.058,Z 705.322,A -85,B 0,C 180,E1 17855.668,E2 17855.668} C_VEL
LIN {X 0,Y 296.652,Z 725.146,A -85,B 0,C 180,E1 17859.802,E2 17859.802} C_VEL
LIN {X 0,Y 284.775,Z 758.696,A -85,B 0,C 180,E1 17863.448,E2 17863.448} C_VEL
LIN {X 0,Y 271.483,Z 788.953,A -85,B 0,C 180,E1 17868.41,E2 17868.41} C_VEL
LIN {X 0,Y 259.544,Z 813.42,A -85,B 0,C 180,E1 17874.313,E2 17874.313} C_VEL
LIN {X 0,Y 248.976,Z 834.79,A -85,B 0,C 180,E1 17882.009,E2 17882.009} C_VEL
LIN {X 0,Y 242.287,Z 849.81,A -85,B 0,C 180,E1 17890.425,E2 17890.425} C_VEL
LIN {X 0,Y 239.444,Z 859.16,A -85,B 0,C 180,E1 17899.065,E2 17899.065} C_VEL
LIN {X 0,Y 238.849,Z 862.842,A -85,B 0,C 180,E1 17906.366,E2 17906.366} C_VEL
LIN {X 0,Y 239.039,Z 863.306,A -85,B 0,C 180,E1 17910,E2 17910} C_VEL
LIN {X 0,Y 239.037,Z 861.467,A -85,B 0,C 180,E1 17917.278,E2 17917.278} C_VEL
LIN {X 0,Y 240.564,Z 854.867,A -85,B 0,C 180,E1 17925.515,E2 17925.515} C_VEL
LIN {X 0,Y 245.725,Z 841.784,A -85,B 0,C 180,E1 17934.576,E2 17934.576} C_VEL
LIN {X 0,Y 255.286,Z 821.943,A -85,B 0,C 180,E1 17942.992,E2 17942.992} C_VEL
LIN {X 0,Y 266.914,Z 798.444,A -85,B 0,C 180,E1 17949.559,E2 17949.559} C_VEL
LIN {X 0,Y 279.586,Z 771.163,A -85,B 0,C 180,E1 17954.748,E2 17954.748} C_VEL
LIN {X 0,Y 292.105,Z 739.027,A -85,B 0,C 180,E1 17958.853,E2 17958.853} C_VEL
LIN {X 0,Y 296.631,Z 725.102,A -85,B 0,C 180,E1 17960.21,E2 17960.21} C_VEL
LIN {X 0,Y 290.978,Z 701.846,A -85,B 0,C 180,E1 17965.093,E2 17965.093} C_VEL
LIN {X 0,Y 281.369,Z 677.048,A -85,B 0,C 180,E1 17971.501,E2 17971.501} C_VEL
LIN {X 0,Y 272.264,Z 660.019,A -85,B 0,C 180,E1 17977.53,E2 17977.53} C_VEL
LIN {X 0,Y 264.97,Z 648.146,A -85,B 0,C 180,E1 17983.406,E2 17983.406} C_VEL
LIN {X 0,Y 261.168,Z 641.898,A -85,B 0,C 180,E1 17987.451,E2 17987.451} C_VEL
LIN {X 0,Y 257.73,Z 636.034,A -85,B 0,C 180,E1 17992.835,E2 17992.835} C_VEL
LIN {X 0,Y 255.863,Z 634.217,A -85,B 0,C 180,E1 18000.961,E2 18000.961} C_VEL
LIN {X 0,Y 255.936,Z 637.047,A -85,B 0,C 180,E1 18003.835,E2 18003.835} C_VEL
LIN {X 0,Y 256.57,Z 645.567,A -85,B 0,C 180,E1 18008.454,E2 18008.454} C_VEL
LIN {X 0,Y 260.152,Z 651.403,A -85,B 0,C 180,E1 18014.004,E2 18014.004} C_VEL
LIN {X 0,Y 264.692,Z 659.692,A -85,B 0,C 180,E1 18018.991,E2 18018.991} C_VEL
LIN {X 0,Y 274.12,Z 677.481,A -85,B 0,C 180,E1 18026.823,E2 18026.823} C_VEL
LIN {X 0,Y 288.793,Z 696.385,A -85,B 0,C 180,E1 18035.224,E2 18035.224} C_VEL
LIN {X 0,Y 300.752,Z 708.783,A -85,B 0,C 180,E1 18041.997,E2 18041.997} C_VEL
LIN {X 0,Y 310.665,Z 719.857,A -85,B 0,C 180,E1 18048.397,E2 18048.397} C_VEL
LIN {X 0,Y 318.465,Z 728.039,A -85,B 0,C 180,E1 18053.927,E2 18053.927} C_VEL
LIN {X 0,Y 325.367,Z 734.526,A -85,B 0,C 180,E1 18059.211,E2 18059.211} C_VEL
LIN {X 0,Y 331.092,Z 740.147,A -85,B 0,C 180,E1 18064.43,E2 18064.43} C_VEL
LIN {X 0,Y 335.107,Z 744.415,A -85,B 0,C 180,E1 18068.811,E2 18068.811} C_VEL
LIN {X 0,Y 339.343,Z 748.466,A -85,B 0,C 180,E1 18074.472,E2 18074.472} C_VEL
LIN {X 0,Y 342.883,Z 750.041,A -85,B 0,C 180,E1 18079.827,E2 18079.827} C_VEL
LIN {X 0,Y 344.611,Z 751.224,A -85,B 0,C 180,E1 18084.959,E2 18084.959} C_VEL
LIN {X 0,Y 345.094,Z 751.853,A -85,B 0,C 180,E1 18090,E2 18090} C_VEL
LIN {X 0,Y 344.728,Z 751.146,A -85,B 0,C 180,E1 18095.039,E2 18095.039} C_VEL
LIN {X 0,Y 342.861,Z 749.979,A -85,B 0,C 180,E1 18100.174,E2 18100.174} C_VEL
LIN {X 0,Y 339.361,Z 748.494,A -85,B 0,C 180,E1 18105.527,E2 18105.527} C_VEL
LIN {X 0,Y 335.095,Z 744.37,A -85,B 0,C 180,E1 18111.19,E2 18111.19} C_VEL
LIN {X 0,Y 331.132,Z 740.152,A -85,B 0,C 180,E1 18115.582,E2 18115.582} C_VEL
LIN {X 0,Y 324.712,Z 733.549,A -85,B 0,C 180,E1 18121.401,E2 18121.401} C_VEL
LIN {X 0,Y 316.826,Z 725.648,A -85,B 0,C 180,E1 18127.439,E2 18127.439} C_VEL
LIN {X 0,Y 308.013,Z 716.348,A -85,B 0,C 180,E1 18133.486,E2 18133.486} C_VEL
LIN {X 0,Y 297.791,Z 705.957,A -85,B 0,C 180,E1 18139.698,E2 18139.698} C_VEL
LIN {X 0,Y 286.122,Z 693.423,A -85,B 0,C 180,E1 18146.241,E2 18146.241} C_VEL
LIN {X 0,Y 269.411,Z 668.44,A -85,B 0,C 180,E1 18156.829,E2 18156.829} C_VEL
LIN {X 0,Y 262.639,Z 655.749,A -85,B 0,C 180,E1 18163.134,E2 18163.134} C_VEL
LIN {X 0,Y 258.825,Z 649.209,A -85,B 0,C 180,E1 18167.752,E2 18167.752} C_VEL
LIN {X 0,Y 256.17,Z 643.368,A -85,B 0,C 180,E1 18172.992,E2 18172.992} C_VEL
LIN {X 0,Y 254.91,Z 642.24,A -85,B 0,C 180,E1 18182.547,E2 18182.547} C_VEL
LIN {X 0,Y 256.349,Z 643.834,A -85,B 0,C 180,E1 18186.884,E2 18186.884} C_VEL
LIN {X 0,Y 259.752,Z 649.738,A -85,B 0,C 180,E1 18192.619,E2 18192.619} C_VEL
LIN {X 0,Y 267.394,Z 662.943,A -85,B 0,C 180,E1 18200.285,E2 18200.285} C_VEL
LIN {X 0,Y 276.229,Z 680.899,A -85,B 0,C 180,E1 18207.097,E2 18207.097} C_VEL
LIN {X 0,Y 284.442,Z 702.231,A -85,B 0,C 180,E1 18213.08,E2 18213.08} C_VEL
LIN {X 0,Y 290.184,Z 724.843,A -85,B 0,C 180,E1 18218.243,E2 18218.243} C_VEL
LIN {X 0,Y 290.119,Z 729.908,A -85,B 0,C 180,E1 18219.083,E2 18219.083} C_VEL
LIN {X 0,Y 277.915,Z 761.685,A -85,B 0,C 180,E1 18222.711,E2 18222.711} C_VEL
LIN {X 0,Y 263.941,Z 792.025,A -85,B 0,C 180,E1 18227.918,E2 18227.918} C_VEL
LIN {X 0,Y 250.984,Z 816.986,A -85,B 0,C 180,E1 18234.428,E2 18234.428} C_VEL
LIN {X 0,Y 241.001,Z 836.181,A -85,B 0,C 180,E1 18241.879,E2 18241.879} C_VEL
LIN {X 0,Y 233.977,Z 851.413,A -85,B 0,C 180,E1 18251.122,E2 18251.122} C_VEL
LIN {X 0,Y 231.619,Z 858.924,A -85,B 0,C 180,E1 18258.691,E2 18258.691} C_VEL
LIN {X 0,Y 230.941,Z 862.608,A -85,B 0,C 180,E1 18266.241,E2 18266.241} C_VEL
LIN {X 0,Y 231.135,Z 863.073,A -85,B 0,C 180,E1 18270,E2 18270} C_VEL
LIN {X 0,Y 231.147,Z 861.232,A -85,B 0,C 180,E1 18277.528,E2 18277.528} C_VEL
LIN {X 0,Y 232.842,Z 854.63,A -85,B 0,C 180,E1 18286.043,E2 18286.043} C_VEL
LIN {X 0,Y 238.381,Z 841.544,A -85,B 0,C 180,E1 18295.386,E2 18295.386} C_VEL
LIN {X 0,Y 248.438,Z 821.893,A -85,B 0,C 180,E1 18303.939,E2 18303.939} C_VEL
LIN {X 0,Y 259.986,Z 799.731,A -85,B 0,C 180,E1 18310.337,E2 18310.337} C_VEL
LIN {X 0,Y 273.925,Z 770.925,A -85,B 0,C 180,E1 18315.934,E2 18315.934} C_VEL
LIN {X 0,Y 287.149,Z 738.219,A -85,B 0,C 180,E1 18320.108,E2 18320.108} C_VEL
LIN {X 0,Y 290.499,Z 727.122,A -85,B 0,C 180,E1 18321.295,E2 18321.295} C_VEL
LIN {X 0,Y 285.24,Z 704.514,A -85,B 0,C 180,E1 18326.352,E2 18326.352} C_VEL
LIN {X 0,Y 276.946,Z 682.361,A -85,B 0,C 180,E1 18332.405,E2 18332.405} C_VEL
LIN {X 0,Y 268.95,Z 666.328,A -85,B 0,C 180,E1 18338.326,E2 18338.326} C_VEL
LIN {X 0,Y 262.562,Z 655.308,A -85,B 0,C 180,E1 18344.003,E2 18344.003} C_VEL
LIN {X 0,Y 259.211,Z 649.344,A -85,B 0,C 180,E1 18347.997,E2 18347.997} C_VEL
LIN {X 0,Y 256.234,Z 643.137,A -85,B 0,C 180,E1 18353.539,E2 18353.539} C_VEL
LIN {X 0,Y 254.994,Z 642.291,A -85,B 0,C 180,E1 18363.41,E2 18363.41} C_VEL
LIN {X 0,Y 256.281,Z 643.958,A -85,B 0,C 180,E1 18367.431,E2 18367.431} C_VEL
LIN {X 0,Y 256.57,Z 645.567,A -85,B 0,C 180,E1 18368.454,E2 18368.454} C_VEL
LIN {X 0,Y 257.625,Z 657.599,A -85,B 0,C 180,E1 18373,E2 18373} C_VEL
LIN {X 0,Y 263.737,Z 670.076,A -85,B 0,C 180,E1 18380.322,E2 18380.322} C_VEL
LIN {X 0,Y 279.305,Z 696.321,A -85,B 0,C 180,E1 18391.911,E2 18391.911} C_VEL
LIN {X 0,Y 291.265,Z 709.949,A -85,B 0,C 180,E1 18398.598,E2 18398.598} C_VEL
LIN {X 0,Y 301.359,Z 720.731,A -85,B 0,C 180,E1 18404.703,E2 18404.703} C_VEL
LIN {X 0,Y 311.12,Z 730.795,A -85,B 0,C 180,E1 18411.141,E2 18411.141} C_VEL
LIN {X 0,Y 319.218,Z 738.93,A -85,B 0,C 180,E1 18417.21,E2 18417.21} C_VEL
LIN {X 0,Y 326.775,Z 746.695,A -85,B 0,C 180,E1 18423.903,E2 18423.903} C_VEL
LIN {X 0,Y 331.162,Z 751.095,A -85,B 0,C 180,E1 18428.546,E2 18428.546} C_VEL
LIN {X 0,Y 335.489,Z 755.336,A -85,B 0,C 180,E1 18434.289,E2 18434.289} C_VEL
LIN {X 0,Y 339.065,Z 756.956,A -85,B 0,C 180,E1 18439.711,E2 18439.711} C_VEL
LIN {X 0,Y 340.37,Z 757.247,A -85,B 0,C 180,E1 18442.331,E2 18442.331} C_VEL
LIN {X 0,Y 341.32,Z 758.545,A -85,B 0,C 180,E1 18447.458,E2 18447.458} C_VEL
LIN {X 0,Y 341.268,Z 758.698,A -85,B 0,C 180,E1 18452.543,E2 18452.543} C_VEL
LIN {X 0,Y 340.425,Z 757.255,A -85,B 0,C 180,E1 18457.668,E2 18457.668} C_VEL
LIN {X 0,Y 337.386,Z 756.342,A -85,B 0,C 180,E1 18462.966,E2 18462.966} C_VEL
LIN {X 0,Y 332.69,Z 752.929,A -85,B 0,C 180,E1 18469.407,E2 18469.407} C_VEL
LIN {X 0,Y 328.695,Z 747.859,A -85,B 0,C 180,E1 18474.492,E2 18474.492} C_VEL
LIN {X 0,Y 322.2,Z 742.365,A -85,B 0,C 180,E1 18480.209,E2 18480.209} C_VEL
LIN {X 0,Y 314.742,Z 734.942,A -85,B 0,C 180,E1 18486.109,E2 18486.109} C_VEL
LIN {X 0,Y 306.226,Z 725.992,A -85,B 0,C 180,E1 18492.124,E2 18492.124} C_VEL
LIN {X 0,Y 296.414,Z 715.277,A -85,B 0,C 180,E1 18498.387,E2 18498.387} C_VEL
LIN {X 0,Y 284.578,Z 702.978,A -85,B 0,C 180,E1 18505.109,E2 18505.109} C_VEL
LIN {X 0,Y 266.87,Z 677.193,A -85,B 0,C 180,E1 18516.595,E2 18516.595} C_VEL
LIN {X 0,Y 260.609,Z 663.473,A -85,B 0,C 180,E1 18523.107,E2 18523.107} C_VEL
LIN {X 0,Y 256.662,Z 656.569,A -85,B 0,C 180,E1 18528.295,E2 18528.295} C_VEL
LIN {X 0,Y 254.201,Z 650.547,A -85,B 0,C 180,E1 18534.011,E2 18534.011} C_VEL
LIN {X 0,Y 253.834,Z 650.296,A -85,B 0,C 180,E1 18544.27,E2 18544.27} C_VEL
LIN {X 0,Y 254.702,Z 651.977,A -85,B 0,C 180,E1 18546.929,E2 18546.929} C_VEL
LIN {X 0,Y 258.464,Z 659.138,A -85,B 0,C 180,E1 18553.329,E2 18553.329} C_VEL
LIN {X 0,Y 264.541,Z 670.17,A -85,B 0,C 180,E1 18559.859,E2 18559.859} C_VEL
LIN {X 0,Y 272.835,Z 688.12,A -85,B 0,C 180,E1 18566.837,E2 18566.837} C_VEL
LIN {X 0,Y 280.247,Z 709.803,A -85,B 0,C 180,E1 18573.022,E2 18573.022} C_VEL
LIN {X 0,Y 284.619,Z 730.215,A -85,B 0,C 180,E1 18577.798,E2 18577.798} C_VEL
LIN {X 0,Y 272.543,Z 761.437,A -85,B 0,C 180,E1 18581.47,E2 18581.47} C_VEL
LIN {X 0,Y 258.347,Z 791.076,A -85,B 0,C 180,E1 18586.567,E2 18586.567} C_VEL
LIN {X 0,Y 244.726,Z 816.226,A -85,B 0,C 180,E1 18593.158,E2 18593.158} C_VEL
LIN {X 0,Y 233.836,Z 836.065,A -85,B 0,C 180,E1 18601.01,E2 18601.01} C_VEL
LIN {X 0,Y 226.355,Z 851.174,A -85,B 0,C 180,E1 18610.461,E2 18610.461} C_VEL
LIN {X 0,Y 223.782,Z 858.688,A -85,B 0,C 180,E1 18618.289,E2 18618.289} C_VEL
LIN {X 0,Y 223.049,Z 862.374,A -85,B 0,C 180,E1 18626.108,E2 18626.108} C_VEL
LIN {X 0,Y 223.231,Z 862.839,A -85,B 0,C 180,E1 18630,E2 18630} C_VEL
LIN {X 0,Y 223.261,Z 860.997,A -85,B 0,C 180,E1 18637.795,E2 18637.795} C_VEL
LIN {X 0,Y 225.144,Z 854.393,A -85,B 0,C 180,E1 18646.607,E2 18646.607} C_VEL
LIN {X 0,Y 231.1,Z 841.305,A -85,B 0,C 180,E1 18656.246,E2 18656.246} C_VEL
LIN {X 0,Y 241.521,Z 822.056,A -85,B 0,C 180,E1 18664.863,E2 18664.863} C_VEL
